LIN {X 101.752,Y 87.486,Z 76.388,A 180.000,B 0.000,C 180.000} C_DIS
LIN {X 101.682,Y 87.454,Z 76.385,A 180.000,B 0.000,C 180.000} C_DIS
LIN {X 101.612,Y 87.423,Z 76.382,A 180.000,B 0.000,C 180.000} C_DIS
LIN {X 101.541,Y 87.395,Z 76.380,A 180.000,B 0.000,C 180.000} C_DIS
LIN {X 101.323,Y 87.307,Z 76.371,A 180.000,B 0.000,C 180.000} C_DIS
LIN {X 101.250,Y 87.278,Z 76.369,A 180.000,B 0.000,C 180.000} C_DIS
LIN {X 101.178,Y 87.250,Z 76.366,A 180.000,B 0.000,C 180.000} C_DIS
LIN {X 101.106,Y 87.223,Z 76.363,A 180.000,B 0.000,C 180.000} C_DIS
LIN {X 101.033,Y 87.198,Z 76.361,A 180.000,B 0.000,C 180.000} C_DIS
LIN {X 100.961,Y 87.173,Z 76.358,A 180.000,B 0.000,C 180.000} C_DIS
LIN {X 100.886,Y 87.148,Z 76.355,A 180.000,B 0.000,C 180.000} C_DIS
LIN {X 100.591,Y 87.048,Z 76.344,A 180.000,B 0.000,C 180.000} C_DIS
LIN {X 100.518,Y 87.024,Z 76.342,A 180.000,B 0.000,C 180.000} C_DIS
LIN {X 100.445,Y 87.002,Z 76.339,A 180.000,B 0.000,C 180.000} C_DIS
LIN {X 100.371,Y 86.981,Z 76.336,A 180.000,B 0.000,C 180.000} C_DIS
LIN {X 100.220,Y 86.940,Z 76.331,A 180.000,B 0.000,C 180.000} C_DIS
LIN {X 100.070,Y 86.898,Z 76.325,A 180.000,B 0.000,C 180.000} C_DIS
LIN {X 99.995,Y 86.878,Z 76.323,A 180.000,B 0.000,C 180.000} C_DIS
LIN {X 99.920,Y 86.860,Z 76.320,A 180.000,B 0.000,C 180.000} C_DIS
LIN {X 99.845,Y 86.843,Z 76.317,A 180.000,B 0.000,C 180.000} C_DIS
LIN {X 99.769,Y 86.827,Z 76.315,A 180.000,B 0.000,C 180.000} C_DIS
LIN {X 99.615,Y 86.794,Z 76.309,A 180.000,B 0.000,C 180.000} C_DIS
LIN {X 99.539,Y 86.777,Z 76.306,A 180.000,B 0.000,C 180.000} C_DIS
LIN {X 99.462,Y 86.760,Z 76.304,A 180.000,B 0.000,C 180.000} C_DIS
LIN {X 99.386,Y 86.745,Z 76.301,A 180.000,B 0.000,C 180.000} C_DIS
LIN {X 99.311,Y 86.729,Z 76.298,A 180.000,B 0.000,C 180.000} C_DIS
LIN {X 99.235,Y 86.716,Z 76.295,A 180.000,B 0.000,C 180.000} C_DIS
LIN {X 99.159,Y 86.703,Z 76.293,A 180.000,B 0.000,C 180.000} C_DIS
LIN {X 99.004,Y 86.679,Z 76.287,A 180.000,B 0.000,C 180.000} C_DIS
LIN {X 98.848,Y 86.654,Z 76.282,A 180.000,B 0.000,C 180.000} C_DIS
LIN {X 98.772,Y 86.643,Z 76.279,A 180.000,B 0.000,C 180.000} C_DIS
LIN {X 98.696,Y 86.633,Z 76.276,A 180.000,B 0.000,C 180.000} C_DIS
LIN {X 98.619,Y 86.625,Z 76.274,A 180.000,B 0.000,C 180.000} C_DIS
LIN {X 98.543,Y 86.617,Z 76.271,A 180.000,B 0.000,C 180.000} C_DIS
LIN {X 98.386,Y 86.602,Z 76.266,A 180.000,B 0.000,C 180.000} C_DIS
LIN {X 98.308,Y 86.594,Z 76.263,A 180.000,B 0.000,C 180.000} C_DIS
LIN {X 98.230,Y 86.586,Z 76.260,A 180.000,B 0.000,C 180.000} C_DIS
LIN {X 98.153,Y 86.580,Z 76.257,A 180.000,B 0.000,C 180.000} C_DIS
LIN {X 98.076,Y 86.574,Z 76.255,A 180.000,B 0.000,C 180.000} C_DIS
LIN {X 97.999,Y 86.569,Z 76.252,A 180.000,B 0.000,C 180.000} C_DIS
LIN {X 97.921,Y 86.565,Z 76.249,A 180.000,B 0.000,C 180.000} C_DIS
LIN {X 97.765,Y 86.558,Z 76.244,A 180.000,B 0.000,C 180.000} C_DIS
LIN {X 97.608,Y 86.551,Z 76.238,A 180.000,B 0.000,C 180.000} C_DIS
LIN {X 97.531,Y 86.548,Z 76.236,A 180.000,B 0.000,C 180.000} C_DIS
LIN {X 97.453,Y 86.547,Z 76.233,A 180.000,B 0.000,C 180.000} C_DIS
LIN {X 97.375,Y 86.548,Z 76.230,A 180.000,B 0.000,C 180.000} C_DIS
LIN {X 97.298,Y 86.549,Z 76.228,A 180.000,B 0.000,C 180.000} C_DIS
LIN {X 97.141,Y 86.551,Z 76.222,A 180.000,B 0.000,C 180.000} C_DIS
LIN {X 97.063,Y 86.552,Z 76.219,A 180.000,B 0.000,C 180.000} C_DIS
LIN {X 96.984,Y 86.553,Z 76.217,A 180.000,B 0.000,C 180.000} C_DIS
LIN {X 96.906,Y 86.556,Z 76.214,A 180.000,B 0.000,C 180.000} C_DIS
LIN {X 96.829,Y 86.559,Z 76.211,A 180.000,B 0.000,C 180.000} C_DIS
LIN {X 96.751,Y 86.563,Z 76.208,A 180.000,B 0.000,C 180.000} C_DIS
LIN {X 96.674,Y 86.568,Z 76.206,A 180.000,B 0.000,C 180.000} C_DIS
LIN {X 96.518,Y 86.579,Z 76.200,A 180.000,B 0.000,C 180.000} C_DIS
LIN {X 96.361,Y 86.590,Z 76.195,A 180.000,B 0.000,C 180.000} C_DIS
LIN {X 96.284,Y 86.595,Z 76.192,A 180.000,B 0.000,C 180.000} C_DIS
LIN {X 96.206,Y 86.603,Z 76.189,A 180.000,B 0.000,C 180.000} C_DIS
LIN {X 96.129,Y 86.613,Z 76.187,A 180.000,B 0.000,C 180.000} C_DIS
LIN {X 95.973,Y 86.632,Z 76.181,A 180.000,B 0.000,C 180.000} C_DIS
LIN {X 95.895,Y 86.642,Z 76.179,A 180.000,B 0.000,C 180.000} C_DIS
LIN {X 95.818,Y 86.652,Z 76.176,A 180.000,B 0.000,C 180.000} C_DIS
LIN {X 95.740,Y 86.662,Z 76.173,A 180.000,B 0.000,C 180.000} C_DIS
LIN {X 95.663,Y 86.674,Z 76.171,A 180.000,B 0.000,C 180.000} C_DIS
LIN {X 95.586,Y 86.687,Z 76.168,A 180.000,B 0.000,C 180.000} C_DIS
LIN {X 95.509,Y 86.701,Z 76.166,A 180.000,B 0.000,C 180.000} C_DIS
LIN {X 95.355,Y 86.729,Z 76.160,A 180.000,B 0.000,C 180.000} C_DIS
LIN {X 95.278,Y 86.743,Z 76.158,A 180.000,B 0.000,C 180.000} C_DIS
LIN {X 95.200,Y 86.757,Z 76.155,A 180.000,B 0.000,C 180.000} C_DIS
LIN {X 95.123,Y 86.771,Z 76.153,A 180.000,B 0.000,C 180.000} C_DIS
LIN {X 94.970,Y 86.803,Z 76.148,A 180.000,B 0.000,C 180.000} C_DIS
LIN {X 94.819,Y 86.839,Z 76.143,A 180.000,B 0.000,C 180.000} C_DIS
LIN {X 94.667,Y 86.876,Z 76.138,A 180.000,B 0.000,C 180.000} C_DIS
LIN {X 94.514,Y 86.914,Z 76.133,A 180.000,B 0.000,C 180.000} C_DIS
LIN {X 94.364,Y 86.957,Z 76.128,A 180.000,B 0.000,C 180.000} C_DIS
LIN {X 94.214,Y 87.002,Z 76.124,A 180.000,B 0.000,C 180.000} C_DIS
LIN {X 94.064,Y 87.048,Z 76.119,A 180.000,B 0.000,C 180.000} C_DIS
LIN {X 93.913,Y 87.094,Z 76.115,A 180.000,B 0.000,C 180.000} C_DIS
LIN {X 93.765,Y 87.143,Z 76.110,A 180.000,B 0.000,C 180.000} C_DIS
LIN {X 93.618,Y 87.197,Z 76.106,A 180.000,B 0.000,C 180.000} C_DIS
LIN {X 93.471,Y 87.251,Z 76.102,A 180.000,B 0.000,C 180.000} C_DIS
LIN {X 93.325,Y 87.305,Z 76.097,A 180.000,B 0.000,C 180.000} C_DIS
LIN {X 93.180,Y 87.366,Z 76.093,A 180.000,B 0.000,C 180.000} C_DIS
LIN {X 93.035,Y 87.429,Z 76.089,A 180.000,B 0.000,C 180.000} C_DIS
LIN {X 92.891,Y 87.491,Z 76.085,A 180.000,B 0.000,C 180.000} C_DIS
LIN {X 92.748,Y 87.555,Z 76.081,A 180.000,B 0.000,C 180.000} C_DIS
LIN {X 92.606,Y 87.622,Z 76.077,A 180.000,B 0.000,C 180.000} C_DIS
LIN {X 92.465,Y 87.692,Z 76.073,A 180.000,B 0.000,C 180.000} C_DIS
LIN {X 92.325,Y 87.763,Z 76.070,A 180.000,B 0.000,C 180.000} C_DIS
LIN {X 92.185,Y 87.834,Z 76.066,A 180.000,B 0.000,C 180.000} C_DIS
LIN {X 92.048,Y 87.911,Z 76.063,A 180.000,B 0.000,C 180.000} C_DIS
LIN {X 91.912,Y 87.989,Z 76.059,A 180.000,B 0.000,C 180.000} C_DIS
LIN {X 91.776,Y 88.068,Z 76.056,A 180.000,B 0.000,C 180.000} C_DIS
LIN {X 91.641,Y 88.148,Z 76.052,A 180.000,B 0.000,C 180.000} C_DIS
LIN {X 91.508,Y 88.232,Z 76.049,A 180.000,B 0.000,C 180.000} C_DIS
LIN {X 91.376,Y 88.318,Z 76.046,A 180.000,B 0.000,C 180.000} C_DIS
LIN {X 91.245,Y 88.404,Z 76.043,A 180.000,B 0.000,C 180.000} C_DIS
LIN {X 91.113,Y 88.491,Z 76.040,A 180.000,B 0.000,C 180.000} C_DIS
LIN {X 90.986,Y 88.583,Z 76.037,A 180.000,B 0.000,C 180.000} C_DIS
LIN {X 90.860,Y 88.677,Z 76.035,A 180.000,B 0.000,C 180.000} C_DIS
LIN {X 90.734,Y 88.770,Z 76.032,A 180.000,B 0.000,C 180.000} C_DIS
LIN {X 90.609,Y 88.866,Z 76.029,A 180.000,B 0.000,C 180.000} C_DIS
LIN {X 90.366,Y 89.066,Z 76.025,A 180.000,B 0.000,C 180.000} C_DIS
LIN {X 90.125,Y 89.268,Z 76.020,A 180.000,B 0.000,C 180.000} C_DIS
LIN {X 89.894,Y 89.482,Z 76.016,A 180.000,B 0.000,C 180.000} C_DIS
LIN {X 89.666,Y 89.700,Z 76.013,A 180.000,B 0.000,C 180.000} C_DIS
LIN {X 89.449,Y 89.927,Z 76.009,A 180.000,B 0.000,C 180.000} C_DIS
LIN {X 89.232,Y 90.156,Z 76.007,A 180.000,B 0.000,C 180.000} C_DIS
LIN {X 89.028,Y 90.395,Z 76.004,A 180.000,B 0.000,C 180.000} C_DIS
LIN {X 88.826,Y 90.638,Z 76.003,A 180.000,B 0.000,C 180.000} C_DIS
LIN {X 88.637,Y 90.889,Z 76.001,A 180.000,B 0.000,C 180.000} C_DIS
LIN {X 88.449,Y 91.142,Z 76.000,A 180.000,B 0.000,C 180.000} C_DIS
LIN {X 88.273,Y 91.403,Z 76.000,A 180.000,B 0.000,C 180.000} C_DIS
LIN {X 88.220,Y 91.484,Z 76.000,A 180.000,B 0.000,C 180.000} C_DIS
; Cutting Move Starts
LIN {X 88.186,Y 91.533,Z 76.000,A 180.000,B 0.000,C 180.000} C_DIS
LIN {X 88.137,Y 91.609,Z 76.000,A 180.000,B 0.000,C 180.000} C_DIS
LIN {X 88.075,Y 91.712,Z 76.000,A 180.000,B 0.000,C 180.000} C_DIS
LIN {X 87.958,Y 91.910,Z 76.000,A 180.000,B 0.000,C 180.000} C_DIS
LIN {X 87.864,Y 92.070,Z 76.000,A 180.000,B 0.000,C 180.000} C_DIS
LIN {X 87.779,Y 92.224,Z 76.000,A 180.000,B 0.000,C 180.000} C_DIS
LIN {X 87.766,Y 92.249,Z 76.000,A 180.000,B 0.000,C 180.000} C_DIS
LIN {X 87.674,Y 92.427,Z 76.000,A 180.000,B 0.000,C 180.000} C_DIS
LIN {X 87.581,Y 92.606,Z 76.000,A 180.000,B 0.000,C 180.000} C_DIS
LIN {X 87.494,Y 92.785,Z 76.000,A 180.000,B 0.000,C 180.000} C_DIS
LIN {X 87.334,Y 93.142,Z 76.000,A 180.000,B 0.000,C 180.000} C_DIS
LIN {X 87.260,Y 93.321,Z 76.000,A 180.000,B 0.000,C 180.000} C_DIS
LIN {X 87.243,Y 93.365,Z 76.000,A 180.000,B 0.000,C 180.000} C_DIS
LIN {X 87.191,Y 93.500,Z 76.000,A 180.000,B 0.000,C 180.000} C_DIS
LIN {X 87.123,Y 93.679,Z 76.000,A 180.000,B 0.000,C 180.000} C_DIS
LIN {X 87.064,Y 93.833,Z 76.000,A 180.000,B 0.000,C 180.000} C_DIS
LIN {X 87.055,Y 93.857,Z 76.000,A 180.000,B 0.000,C 180.000} C_DIS
LIN {X 86.997,Y 94.036,Z 76.000,A 180.000,B 0.000,C 180.000} C_DIS
LIN {X 86.940,Y 94.215,Z 76.000,A 180.000,B 0.000,C 180.000} C_DIS
LIN {X 86.885,Y 94.388,Z 76.000,A 180.000,B 0.000,C 180.000} C_DIS
LIN {X 86.884,Y 94.394,Z 76.000,A 180.000,B 0.000,C 180.000} C_DIS
LIN {X 86.836,Y 94.573,Z 76.000,A 180.000,B 0.000,C 180.000} C_DIS
LIN {X 86.790,Y 94.751,Z 76.000,A 180.000,B 0.000,C 180.000} C_DIS
LIN {X 86.744,Y 94.930,Z 76.000,A 180.000,B 0.000,C 180.000} C_DIS
LIN {X 86.707,Y 95.079,Z 76.000,A 180.000,B 0.000,C 180.000} C_DIS
LIN {X 86.700,Y 95.109,Z 76.000,A 180.000,B 0.000,C 180.000} C_DIS
LIN {X 86.664,Y 95.288,Z 76.000,A 180.000,B 0.000,C 180.000} C_DIS
LIN {X 86.629,Y 95.466,Z 76.000,A 180.000,B 0.000,C 180.000} C_DIS
LIN {X 86.595,Y 95.645,Z 76.000,A 180.000,B 0.000,C 180.000} C_DIS
LIN {X 86.569,Y 95.824,Z 76.000,A 180.000,B 0.000,C 180.000} C_DIS
LIN {X 86.528,Y 96.116,Z 76.000,A 180.000,B 0.000,C 180.000} C_DIS
LIN {X 86.519,Y 96.181,Z 76.000,A 180.000,B 0.000,C 180.000} C_DIS
LIN {X 86.498,Y 96.360,Z 76.000,A 180.000,B 0.000,C 180.000} C_DIS
LIN {X 86.483,Y 96.539,Z 76.000,A 180.000,B 0.000,C 180.000} C_DIS
LIN {X 86.468,Y 96.718,Z 76.000,A 180.000,B 0.000,C 180.000} C_DIS
LIN {X 86.455,Y 96.897,Z 76.000,A 180.000,B 0.000,C 180.000} C_DIS
LIN {X 86.449,Y 97.075,Z 76.000,A 180.000,B 0.000,C 180.000} C_DIS
LIN {X 86.444,Y 97.254,Z 76.000,A 180.000,B 0.000,C 180.000} C_DIS
LIN {X 86.440,Y 97.433,Z 76.000,A 180.000,B 0.000,C 180.000} C_DIS
LIN {X 86.440,Y 97.612,Z 76.000,A 180.000,B 0.000,C 180.000} C_DIS
LIN {X 86.445,Y 97.790,Z 76.000,A 180.000,B 0.000,C 180.000} C_DIS
LIN {X 86.450,Y 97.969,Z 76.000,A 180.000,B 0.000,C 180.000} C_DIS
LIN {X 86.457,Y 98.148,Z 76.000,A 180.000,B 0.000,C 180.000} C_DIS
LIN {X 86.472,Y 98.327,Z 76.000,A 180.000,B 0.000,C 180.000} C_DIS
LIN {X 86.487,Y 98.505,Z 76.000,A 180.000,B 0.000,C 180.000} C_DIS
LIN {X 86.503,Y 98.684,Z 76.000,A 180.000,B 0.000,C 180.000} C_DIS
LIN {X 86.525,Y 98.863,Z 76.000,A 180.000,B 0.000,C 180.000} C_DIS
LIN {X 86.528,Y 98.884,Z 76.000,A 180.000,B 0.000,C 180.000} C_DIS
LIN {X 86.575,Y 99.221,Z 76.000,A 180.000,B 0.000,C 180.000} C_DIS
LIN {X 86.603,Y 99.399,Z 76.000,A 180.000,B 0.000,C 180.000} C_DIS
LIN {X 86.638,Y 99.578,Z 76.000,A 180.000,B 0.000,C 180.000} C_DIS
LIN {X 86.673,Y 99.757,Z 76.000,A 180.000,B 0.000,C 180.000} C_DIS
LIN {X 86.707,Y 99.921,Z 76.000,A 180.000,B 0.000,C 180.000} C_DIS
LIN {X 86.710,Y 99.936,Z 76.000,A 180.000,B 0.000,C 180.000} C_DIS
LIN {X 86.755,Y 100.114,Z 76.000,A 180.000,B 0.000,C 180.000} C_DIS
LIN {X 86.848,Y 100.472,Z 76.000,A 180.000,B 0.000,C 180.000} C_DIS
LIN {X 86.885,Y 100.612,Z 76.000,A 180.000,B 0.000,C 180.000} C_DIS
LIN {X 86.897,Y 100.651,Z 76.000,A 180.000,B 0.000,C 180.000} C_DIS
LIN {X 86.954,Y 100.829,Z 76.000,A 180.000,B 0.000,C 180.000} C_DIS
LIN {X 87.011,Y 101.008,Z 76.000,A 180.000,B 0.000,C 180.000} C_DIS
LIN {X 87.064,Y 101.167,Z 76.000,A 180.000,B 0.000,C 180.000} C_DIS
LIN {X 87.071,Y 101.187,Z 76.000,A 180.000,B 0.000,C 180.000} C_DIS
LIN {X 87.140,Y 101.366,Z 76.000,A 180.000,B 0.000,C 180.000} C_DIS
LIN {X 87.208,Y 101.545,Z 76.000,A 180.000,B 0.000,C 180.000} C_DIS
LIN {X 87.243,Y 101.635,Z 76.000,A 180.000,B 0.000,C 180.000} C_DIS
LIN {X 87.278,Y 101.723,Z 76.000,A 180.000,B 0.000,C 180.000} C_DIS
LIN {X 87.354,Y 101.902,Z 76.000,A 180.000,B 0.000,C 180.000} C_DIS
LIN {X 87.434,Y 102.081,Z 76.000,A 180.000,B 0.000,C 180.000} C_DIS
LIN {X 87.515,Y 102.260,Z 76.000,A 180.000,B 0.000,C 180.000} C_DIS
LIN {X 87.601,Y 102.431,Z 76.000,A 180.000,B 0.000,C 180.000} C_DIS
LIN {X 87.697,Y 102.617,Z 76.000,A 180.000,B 0.000,C 180.000} C_DIS
LIN {X 87.779,Y 102.776,Z 76.000,A 180.000,B 0.000,C 180.000} C_DIS
LIN {X 87.790,Y 102.796,Z 76.000,A 180.000,B 0.000,C 180.000} C_DIS
LIN {X 87.890,Y 102.975,Z 76.000,A 180.000,B 0.000,C 180.000} C_DIS
LIN {X 88.101,Y 103.332,Z 76.000,A 180.000,B 0.000,C 180.000} C_DIS
LIN {X 88.137,Y 103.391,Z 76.000,A 180.000,B 0.000,C 180.000} C_DIS
LIN {X 88.216,Y 103.511,Z 76.000,A 180.000,B 0.000,C 180.000} C_DIS
LIN {X 88.336,Y 103.690,Z 76.000,A 180.000,B 0.000,C 180.000} C_DIS
LIN {X 88.457,Y 103.869,Z 76.000,A 180.000,B 0.000,C 180.000} C_DIS
LIN {X 88.494,Y 103.920,Z 76.000,A 180.000,B 0.000,C 180.000} C_DIS
LIN {X 88.588,Y 104.047,Z 76.000,A 180.000,B 0.000,C 180.000} C_DIS
LIN {X 88.722,Y 104.226,Z 76.000,A 180.000,B 0.000,C 180.000} C_DIS
LIN {X 88.852,Y 104.397,Z 76.000,A 180.000,B 0.000,C 180.000} C_DIS
LIN {X 88.858,Y 104.405,Z 76.000,A 180.000,B 0.000,C 180.000} C_DIS
LIN {X 89.007,Y 104.584,Z 76.000,A 180.000,B 0.000,C 180.000} C_DIS
LIN {X 89.158,Y 104.762,Z 76.000,A 180.000,B 0.000,C 180.000} C_DIS
LIN {X 89.209,Y 104.823,Z 76.000,A 180.000,B 0.000,C 180.000} C_DIS
LIN {X 89.319,Y 104.941,Z 76.000,A 180.000,B 0.000,C 180.000} C_DIS
LIN {X 89.388,Y 105.015,Z 76.000,A 180.000,B 0.000,C 180.000} C_DIS
LIN {X 89.567,Y 105.204,Z 76.000,A 180.000,B 0.000,C 180.000} C_DIS
LIN {X 89.656,Y 105.299,Z 76.000,A 180.000,B 0.000,C 180.000} C_DIS
LIN {X 89.746,Y 105.388,Z 76.000,A 180.000,B 0.000,C 180.000} C_DIS
LIN {X 89.925,Y 105.557,Z 76.000,A 180.000,B 0.000,C 180.000} C_DIS
LIN {X 90.030,Y 105.656,Z 76.000,A 180.000,B 0.000,C 180.000} C_DIS
LIN {X 90.103,Y 105.725,Z 76.000,A 180.000,B 0.000,C 180.000} C_DIS
LIN {X 90.232,Y 105.835,Z 76.000,A 180.000,B 0.000,C 180.000} C_DIS
LIN {X 90.461,Y 106.029,Z 76.000,A 180.000,B 0.000,C 180.000} C_DIS
LIN {X 90.640,Y 106.177,Z 76.000,A 180.000,B 0.000,C 180.000} C_DIS
LIN {X 90.660,Y 106.193,Z 76.000,A 180.000,B 0.000,C 180.000} C_DIS
LIN {X 90.818,Y 106.312,Z 76.000,A 180.000,B 0.000,C 180.000} C_DIS
LIN {X 90.997,Y 106.447,Z 76.000,A 180.000,B 0.000,C 180.000} C_DIS
LIN {X 91.140,Y 106.550,Z 76.000,A 180.000,B 0.000,C 180.000} C_DIS
LIN {X 91.176,Y 106.574,Z 76.000,A 180.000,B 0.000,C 180.000} C_DIS
LIN {X 91.408,Y 106.729,Z 76.000,A 180.000,B 0.000,C 180.000} C_DIS
LIN {X 91.533,Y 106.813,Z 76.000,A 180.000,B 0.000,C 180.000} C_DIS
LIN {X 91.684,Y 106.908,Z 76.000,A 180.000,B 0.000,C 180.000} C_DIS
LIN {X 91.712,Y 106.925,Z 76.000,A 180.000,B 0.000,C 180.000} C_DIS
LIN {X 91.891,Y 107.031,Z 76.000,A 180.000,B 0.000,C 180.000} C_DIS
LIN {X 92.070,Y 107.136,Z 76.000,A 180.000,B 0.000,C 180.000} C_DIS
LIN {X 92.249,Y 107.234,Z 76.000,A 180.000,B 0.000,C 180.000} C_DIS
LIN {X 92.427,Y 107.327,Z 76.000,A 180.000,B 0.000,C 180.000} C_DIS
LIN {X 92.606,Y 107.419,Z 76.000,A 180.000,B 0.000,C 180.000} C_DIS
LIN {X 92.657,Y 107.444,Z 76.000,A 180.000,B 0.000,C 180.000} C_DIS
LIN {X 92.785,Y 107.504,Z 76.000,A 180.000,B 0.000,C 180.000} C_DIS
LIN {X 92.964,Y 107.585,Z 76.000,A 180.000,B 0.000,C 180.000} C_DIS
LIN {X 93.142,Y 107.665,Z 76.000,A 180.000,B 0.000,C 180.000} C_DIS
LIN {X 93.321,Y 107.742,Z 76.000,A 180.000,B 0.000,C 180.000} C_DIS
LIN {X 93.477,Y 107.802,Z 76.000,A 180.000,B 0.000,C 180.000} C_DIS
LIN {X 93.679,Y 107.879,Z 76.000,A 180.000,B 0.000,C 180.000} C_DIS
LIN {X 93.857,Y 107.944,Z 76.000,A 180.000,B 0.000,C 180.000} C_DIS
LIN {X 93.970,Y 107.980,Z 76.000,A 180.000,B 0.000,C 180.000} C_DIS
LIN {X 94.036,Y 108.001,Z 76.000,A 180.000,B 0.000,C 180.000} C_DIS
LIN {X 94.394,Y 108.115,Z 76.000,A 180.000,B 0.000,C 180.000} C_DIS
LIN {X 94.546,Y 108.159,Z 76.000,A 180.000,B 0.000,C 180.000} C_DIS
LIN {X 94.930,Y 108.258,Z 76.000,A 180.000,B 0.000,C 180.000} C_DIS
LIN {X 95.109,Y 108.299,Z 76.000,A 180.000,B 0.000,C 180.000} C_DIS
LIN {X 95.466,Y 108.370,Z 76.000,A 180.000,B 0.000,C 180.000} C_DIS
LIN {X 95.645,Y 108.404,Z 76.000,A 180.000,B 0.000,C 180.000} C_DIS
LIN {X 95.824,Y 108.432,Z 76.000,A 180.000,B 0.000,C 180.000} C_DIS
LIN {X 96.181,Y 108.482,Z 76.000,A 180.000,B 0.000,C 180.000} C_DIS
LIN {X 96.360,Y 108.501,Z 76.000,A 180.000,B 0.000,C 180.000} C_DIS
LIN {X 96.718,Y 108.531,Z 76.000,A 180.000,B 0.000,C 180.000} C_DIS
LIN {X 96.897,Y 108.544,Z 76.000,A 180.000,B 0.000,C 180.000} C_DIS
LIN {X 97.075,Y 108.551,Z 76.000,A 180.000,B 0.000,C 180.000} C_DIS
LIN {X 97.433,Y 108.561,Z 76.000,A 180.000,B 0.000,C 180.000} C_DIS
LIN {X 97.612,Y 108.560,Z 76.000,A 180.000,B 0.000,C 180.000} C_DIS
LIN {X 97.969,Y 108.550,Z 76.000,A 180.000,B 0.000,C 180.000} C_DIS
LIN {X 98.148,Y 108.541,Z 76.000,A 180.000,B 0.000,C 180.000} C_DIS
LIN {X 98.327,Y 108.528,Z 76.000,A 180.000,B 0.000,C 180.000} C_DIS
LIN {X 98.684,Y 108.498,Z 76.000,A 180.000,B 0.000,C 180.000} C_DIS
LIN {X 98.863,Y 108.476,Z 76.000,A 180.000,B 0.000,C 180.000} C_DIS
LIN {X 99.221,Y 108.426,Z 76.000,A 180.000,B 0.000,C 180.000} C_DIS
LIN {X 99.399,Y 108.396,Z 76.000,A 180.000,B 0.000,C 180.000} C_DIS
LIN {X 99.578,Y 108.361,Z 76.000,A 180.000,B 0.000,C 180.000} C_DIS
LIN {X 99.757,Y 108.325,Z 76.000,A 180.000,B 0.000,C 180.000} C_DIS
LIN {X 99.936,Y 108.290,Z 76.000,A 180.000,B 0.000,C 180.000} C_DIS
LIN {X 100.114,Y 108.247,Z 76.000,A 180.000,B 0.000,C 180.000} C_DIS
LIN {X 100.472,Y 108.154,Z 76.000,A 180.000,B 0.000,C 180.000} C_DIS
LIN {X 100.651,Y 108.101,Z 76.000,A 180.000,B 0.000,C 180.000} C_DIS
LIN {X 101.008,Y 107.987,Z 76.000,A 180.000,B 0.000,C 180.000} C_DIS
LIN {X 101.030,Y 107.980,Z 76.000,A 180.000,B 0.000,C 180.000} C_DIS
LIN {X 101.187,Y 107.929,Z 76.000,A 180.000,B 0.000,C 180.000} C_DIS
LIN {X 101.366,Y 107.862,Z 76.000,A 180.000,B 0.000,C 180.000} C_DIS
LIN {X 101.545,Y 107.793,Z 76.000,A 180.000,B 0.000,C 180.000} C_DIS
LIN {X 101.723,Y 107.724,Z 76.000,A 180.000,B 0.000,C 180.000} C_DIS
LIN {X 101.902,Y 107.645,Z 76.000,A 180.000,B 0.000,C 180.000} C_DIS
LIN {X 102.081,Y 107.565,Z 76.000,A 180.000,B 0.000,C 180.000} C_DIS
LIN {X 102.260,Y 107.483,Z 76.000,A 180.000,B 0.000,C 180.000} C_DIS
LIN {X 102.343,Y 107.444,Z 76.000,A 180.000,B 0.000,C 180.000} C_DIS
LIN {X 102.438,Y 107.396,Z 76.000,A 180.000,B 0.000,C 180.000} C_DIS
LIN {X 102.692,Y 107.265,Z 76.000,A 180.000,B 0.000,C 180.000} C_DIS
LIN {X 102.796,Y 107.211,Z 76.000,A 180.000,B 0.000,C 180.000} C_DIS
LIN {X 102.975,Y 107.110,Z 76.000,A 180.000,B 0.000,C 180.000} C_DIS
LIN {X 103.153,Y 107.004,Z 76.000,A 180.000,B 0.000,C 180.000} C_DIS
LIN {X 103.316,Y 106.908,Z 76.000,A 180.000,B 0.000,C 180.000} C_DIS
LIN {X 103.332,Y 106.898,Z 76.000,A 180.000,B 0.000,C 180.000} C_DIS
LIN {X 103.511,Y 106.783,Z 76.000,A 180.000,B 0.000,C 180.000} C_DIS
LIN {X 103.690,Y 106.664,Z 76.000,A 180.000,B 0.000,C 180.000} C_DIS
LIN {X 103.860,Y 106.550,Z 76.000,A 180.000,B 0.000,C 180.000} C_DIS
LIN {X 103.869,Y 106.544,Z 76.000,A 180.000,B 0.000,C 180.000} C_DIS
LIN {X 104.047,Y 106.413,Z 76.000,A 180.000,B 0.000,C 180.000} C_DIS
LIN {X 104.226,Y 106.279,Z 76.000,A 180.000,B 0.000,C 180.000} C_DIS
LIN {X 104.340,Y 106.193,Z 76.000,A 180.000,B 0.000,C 180.000} C_DIS
LIN {X 104.405,Y 106.140,Z 76.000,A 180.000,B 0.000,C 180.000} C_DIS
LIN {X 104.557,Y 106.014,Z 76.000,A 180.000,B 0.000,C 180.000} C_DIS
LIN {X 104.715,Y 105.880,Z 76.000,A 180.000,B 0.000,C 180.000} C_DIS
LIN {X 104.768,Y 105.835,Z 76.000,A 180.000,B 0.000,C 180.000} C_DIS
LIN {X 104.941,Y 105.684,Z 76.000,A 180.000,B 0.000,C 180.000} C_DIS
LIN {X 105.160,Y 105.477,Z 76.000,A 180.000,B 0.000,C 180.000} C_DIS
LIN {X 105.299,Y 105.345,Z 76.000,A 180.000,B 0.000,C 180.000} C_DIS
LIN {X 105.344,Y 105.299,Z 76.000,A 180.000,B 0.000,C 180.000} C_DIS
LIN {X 105.513,Y 105.120,Z 76.000,A 180.000,B 0.000,C 180.000} C_DIS
LIN {X 105.656,Y 104.968,Z 76.000,A 180.000,B 0.000,C 180.000} C_DIS
LIN {X 105.681,Y 104.941,Z 76.000,A 180.000,B 0.000,C 180.000} C_DIS
LIN {X 105.835,Y 104.770,Z 76.000,A 180.000,B 0.000,C 180.000} C_DIS
LIN {X 106.014,Y 104.559,Z 76.000,A 180.000,B 0.000,C 180.000} C_DIS
LIN {X 106.142,Y 104.405,Z 76.000,A 180.000,B 0.000,C 180.000} C_DIS
LIN {X 106.193,Y 104.339,Z 76.000,A 180.000,B 0.000,C 180.000} C_DIS
LIN {X 106.412,Y 104.047,Z 76.000,A 180.000,B 0.000,C 180.000} C_DIS
LIN {X 106.543,Y 103.869,Z 76.000,A 180.000,B 0.000,C 180.000} C_DIS
LIN {X 106.550,Y 103.859,Z 76.000,A 180.000,B 0.000,C 180.000} C_DIS
LIN {X 106.664,Y 103.690,Z 76.000,A 180.000,B 0.000,C 180.000} C_DIS
LIN {X 106.784,Y 103.511,Z 76.000,A 180.000,B 0.000,C 180.000} C_DIS
LIN {X 106.899,Y 103.332,Z 76.000,A 180.000,B 0.000,C 180.000} C_DIS
LIN {X 107.110,Y 102.975,Z 76.000,A 180.000,B 0.000,C 180.000} C_DIS
LIN {X 107.210,Y 102.796,Z 76.000,A 180.000,B 0.000,C 180.000} C_DIS
LIN {X 107.265,Y 102.691,Z 76.000,A 180.000,B 0.000,C 180.000} C_DIS
LIN {X 107.396,Y 102.438,Z 76.000,A 180.000,B 0.000,C 180.000} C_DIS
LIN {X 107.444,Y 102.345,Z 76.000,A 180.000,B 0.000,C 180.000} C_DIS
LIN {X 107.485,Y 102.260,Z 76.000,A 180.000,B 0.000,C 180.000} C_DIS
LIN {X 107.566,Y 102.081,Z 76.000,A 180.000,B 0.000,C 180.000} C_DIS
LIN {X 107.646,Y 101.902,Z 76.000,A 180.000,B 0.000,C 180.000} C_DIS
LIN {X 107.722,Y 101.723,Z 76.000,A 180.000,B 0.000,C 180.000} C_DIS
LIN {X 107.792,Y 101.545,Z 76.000,A 180.000,B 0.000,C 180.000} C_DIS
LIN {X 107.860,Y 101.366,Z 76.000,A 180.000,B 0.000,C 180.000} C_DIS
LIN {X 107.929,Y 101.187,Z 76.000,A 180.000,B 0.000,C 180.000} C_DIS
LIN {X 107.980,Y 101.036,Z 76.000,A 180.000,B 0.000,C 180.000} C_DIS
LIN {X 108.046,Y 100.829,Z 76.000,A 180.000,B 0.000,C 180.000} C_DIS
LIN {X 108.103,Y 100.651,Z 76.000,A 180.000,B 0.000,C 180.000} C_DIS
LIN {X 108.152,Y 100.472,Z 76.000,A 180.000,B 0.000,C 180.000} C_DIS
LIN {X 108.245,Y 100.114,Z 76.000,A 180.000,B 0.000,C 180.000} C_DIS
LIN {X 108.290,Y 99.936,Z 76.000,A 180.000,B 0.000,C 180.000} C_DIS
LIN {X 108.327,Y 99.757,Z 76.000,A 180.000,B 0.000,C 180.000} C_DIS
LIN {X 108.362,Y 99.578,Z 76.000,A 180.000,B 0.000,C 180.000} C_DIS
LIN {X 108.397,Y 99.399,Z 76.000,A 180.000,B 0.000,C 180.000} C_DIS
LIN {X 108.425,Y 99.221,Z 76.000,A 180.000,B 0.000,C 180.000} C_DIS
LIN {X 108.450,Y 99.042,Z 76.000,A 180.000,B 0.000,C 180.000} C_DIS
LIN {X 108.475,Y 98.863,Z 76.000,A 180.000,B 0.000,C 180.000} C_DIS
LIN {X 108.497,Y 98.684,Z 76.000,A 180.000,B 0.000,C 180.000} C_DIS
LIN {X 108.513,Y 98.505,Z 76.000,A 180.000,B 0.000,C 180.000} C_DIS
LIN {X 108.528,Y 98.327,Z 76.000,A 180.000,B 0.000,C 180.000} C_DIS
LIN {X 108.543,Y 98.148,Z 76.000,A 180.000,B 0.000,C 180.000} C_DIS
LIN {X 108.550,Y 97.969,Z 76.000,A 180.000,B 0.000,C 180.000} C_DIS
LIN {X 108.555,Y 97.790,Z 76.000,A 180.000,B 0.000,C 180.000} C_DIS
LIN {X 108.560,Y 97.612,Z 76.000,A 180.000,B 0.000,C 180.000} C_DIS
LIN {X 108.560,Y 97.433,Z 76.000,A 180.000,B 0.000,C 180.000} C_DIS
LIN {X 108.556,Y 97.254,Z 76.000,A 180.000,B 0.000,C 180.000} C_DIS
LIN {X 108.551,Y 97.075,Z 76.000,A 180.000,B 0.000,C 180.000} C_DIS
LIN {X 108.545,Y 96.897,Z 76.000,A 180.000,B 0.000,C 180.000} C_DIS
LIN {X 108.532,Y 96.718,Z 76.000,A 180.000,B 0.000,C 180.000} C_DIS
LIN {X 108.517,Y 96.534,Z 76.000,A 180.000,B 0.000,C 180.000} C_DIS
LIN {X 108.502,Y 96.360,Z 76.000,A 180.000,B 0.000,C 180.000} C_DIS
LIN {X 108.481,Y 96.181,Z 76.000,A 180.000,B 0.000,C 180.000} C_DIS
LIN {X 108.456,Y 96.003,Z 76.000,A 180.000,B 0.000,C 180.000} C_DIS
LIN {X 108.431,Y 95.824,Z 76.000,A 180.000,B 0.000,C 180.000} C_DIS
LIN {X 108.405,Y 95.645,Z 76.000,A 180.000,B 0.000,C 180.000} C_DIS
LIN {X 108.371,Y 95.466,Z 76.000,A 180.000,B 0.000,C 180.000} C_DIS
LIN {X 108.336,Y 95.288,Z 76.000,A 180.000,B 0.000,C 180.000} C_DIS
LIN {X 108.300,Y 95.109,Z 76.000,A 180.000,B 0.000,C 180.000} C_DIS
LIN {X 108.256,Y 94.930,Z 76.000,A 180.000,B 0.000,C 180.000} C_DIS
LIN {X 108.210,Y 94.751,Z 76.000,A 180.000,B 0.000,C 180.000} C_DIS
LIN {X 108.159,Y 94.554,Z 76.000,A 180.000,B 0.000,C 180.000} C_DIS
LIN {X 108.116,Y 94.394,Z 76.000,A 180.000,B 0.000,C 180.000} C_DIS
LIN {X 108.060,Y 94.215,Z 76.000,A 180.000,B 0.000,C 180.000} C_DIS
LIN {X 107.980,Y 93.964,Z 76.000,A 180.000,B 0.000,C 180.000} C_DIS
LIN {X 107.945,Y 93.857,Z 76.000,A 180.000,B 0.000,C 180.000} C_DIS
LIN {X 107.877,Y 93.679,Z 76.000,A 180.000,B 0.000,C 180.000} C_DIS
LIN {X 107.802,Y 93.480,Z 76.000,A 180.000,B 0.000,C 180.000} C_DIS
LIN {X 107.740,Y 93.321,Z 76.000,A 180.000,B 0.000,C 180.000} C_DIS
LIN {X 107.666,Y 93.142,Z 76.000,A 180.000,B 0.000,C 180.000} C_DIS
LIN {X 107.506,Y 92.785,Z 76.000,A 180.000,B 0.000,C 180.000} C_DIS
LIN {X 107.444,Y 92.655,Z 76.000,A 180.000,B 0.000,C 180.000} C_DIS
LIN {X 107.419,Y 92.606,Z 76.000,A 180.000,B 0.000,C 180.000} C_DIS
LIN {X 107.265,Y 92.309,Z 76.000,A 180.000,B 0.000,C 180.000} C_DIS
LIN {X 107.234,Y 92.249,Z 76.000,A 180.000,B 0.000,C 180.000} C_DIS
LIN {X 107.136,Y 92.070,Z 76.000,A 180.000,B 0.000,C 180.000} C_DIS
LIN {X 107.086,Y 91.986,Z 76.000,A 180.000,B 0.000,C 180.000} C_DIS
LIN {X 106.908,Y 91.683,Z 76.000,A 180.000,B 0.000,C 180.000} C_DIS
LIN {X 106.814,Y 91.533,Z 76.000,A 180.000,B 0.000,C 180.000} C_DIS
LIN {X 106.694,Y 91.355,Z 76.000,A 180.000,B 0.000,C 180.000} C_DIS
LIN {X 106.574,Y 91.176,Z 76.000,A 180.000,B 0.000,C 180.000} C_DIS
LIN {X 106.550,Y 91.141,Z 76.000,A 180.000,B 0.000,C 180.000} C_DIS
LIN {X 106.446,Y 90.997,Z 76.000,A 180.000,B 0.000,C 180.000} C_DIS
LIN {X 106.371,Y 90.898,Z 76.000,A 180.000,B 0.000,C 180.000} C_DIS
LIN {X 106.193,Y 90.661,Z 76.000,A 180.000,B 0.000,C 180.000} C_DIS
LIN {X 106.177,Y 90.640,Z 76.000,A 180.000,B 0.000,C 180.000} C_DIS
LIN {X 106.030,Y 90.461,Z 76.000,A 180.000,B 0.000,C 180.000} C_DIS
LIN {X 105.835,Y 90.230,Z 76.000,A 180.000,B 0.000,C 180.000} C_DIS
LIN {X 105.723,Y 90.103,Z 76.000,A 180.000,B 0.000,C 180.000} C_DIS
LIN {X 105.656,Y 90.032,Z 76.000,A 180.000,B 0.000,C 180.000} C_DIS
LIN {X 105.555,Y 89.925,Z 76.000,A 180.000,B 0.000,C 180.000} C_DIS
LIN {X 105.386,Y 89.746,Z 76.000,A 180.000,B 0.000,C 180.000} C_DIS
LIN {X 105.299,Y 89.655,Z 76.000,A 180.000,B 0.000,C 180.000} C_DIS
LIN {X 105.207,Y 89.567,Z 76.000,A 180.000,B 0.000,C 180.000} C_DIS
LIN {X 104.941,Y 89.316,Z 76.000,A 180.000,B 0.000,C 180.000} C_DIS
LIN {X 104.821,Y 89.209,Z 76.000,A 180.000,B 0.000,C 180.000} C_DIS
LIN {X 104.584,Y 89.009,Z 76.000,A 180.000,B 0.000,C 180.000} C_DIS
LIN {X 104.405,Y 88.860,Z 76.000,A 180.000,B 0.000,C 180.000} C_DIS
LIN {X 104.396,Y 88.852,Z 76.000,A 180.000,B 0.000,C 180.000} C_DIS
LIN {X 104.226,Y 88.721,Z 76.000,A 180.000,B 0.000,C 180.000} C_DIS
LIN {X 104.047,Y 88.587,Z 76.000,A 180.000,B 0.000,C 180.000} C_DIS
LIN {X 103.924,Y 88.494,Z 76.000,A 180.000,B 0.000,C 180.000} C_DIS
LIN {X 103.869,Y 88.456,Z 76.000,A 180.000,B 0.000,C 180.000} C_DIS
LIN {X 103.690,Y 88.336,Z 76.000,A 180.000,B 0.000,C 180.000} C_DIS
LIN {X 103.511,Y 88.217,Z 76.000,A 180.000,B 0.000,C 180.000} C_DIS
LIN {X 103.387,Y 88.137,Z 76.000,A 180.000,B 0.000,C 180.000} C_DIS
LIN {X 103.332,Y 88.102,Z 76.000,A 180.000,B 0.000,C 180.000} C_DIS
LIN {X 103.153,Y 87.996,Z 76.000,A 180.000,B 0.000,C 180.000} C_DIS
LIN {X 102.975,Y 87.890,Z 76.000,A 180.000,B 0.000,C 180.000} C_DIS
LIN {X 102.796,Y 87.789,Z 76.000,A 180.000,B 0.000,C 180.000} C_DIS
LIN {X 102.778,Y 87.779,Z 76.000,A 180.000,B 0.000,C 180.000} C_DIS
LIN {X 102.432,Y 87.601,Z 76.000,A 180.000,B 0.000,C 180.000} C_DIS
LIN {X 102.260,Y 87.517,Z 76.000,A 180.000,B 0.000,C 180.000} C_DIS
LIN {X 102.081,Y 87.435,Z 76.000,A 180.000,B 0.000,C 180.000} C_DIS
LIN {X 101.902,Y 87.355,Z 76.000,A 180.000,B 0.000,C 180.000} C_DIS
LIN {X 101.723,Y 87.276,Z 76.000,A 180.000,B 0.000,C 180.000} C_DIS
LIN {X 101.640,Y 87.243,Z 76.000,A 180.000,B 0.000,C 180.000} C_DIS
LIN {X 101.366,Y 87.138,Z 76.000,A 180.000,B 0.000,C 180.000} C_DIS
LIN {X 101.187,Y 87.071,Z 76.000,A 180.000,B 0.000,C 180.000} C_DIS
LIN {X 101.166,Y 87.064,Z 76.000,A 180.000,B 0.000,C 180.000} C_DIS
LIN {X 101.008,Y 87.013,Z 76.000,A 180.000,B 0.000,C 180.000} C_DIS
LIN {X 100.609,Y 86.885,Z 76.000,A 180.000,B 0.000,C 180.000} C_DIS
LIN {X 100.472,Y 86.846,Z 76.000,A 180.000,B 0.000,C 180.000} C_DIS
LIN {X 100.114,Y 86.753,Z 76.000,A 180.000,B 0.000,C 180.000} C_DIS
LIN {X 99.936,Y 86.710,Z 76.000,A 180.000,B 0.000,C 180.000} C_DIS
LIN {X 99.917,Y 86.707,Z 76.000,A 180.000,B 0.000,C 180.000} C_DIS
LIN {X 99.578,Y 86.639,Z 76.000,A 180.000,B 0.000,C 180.000} C_DIS
LIN {X 99.399,Y 86.604,Z 76.000,A 180.000,B 0.000,C 180.000} C_DIS
LIN {X 99.221,Y 86.574,Z 76.000,A 180.000,B 0.000,C 180.000} C_DIS
LIN {X 98.863,Y 86.524,Z 76.000,A 180.000,B 0.000,C 180.000} C_DIS
LIN {X 98.684,Y 86.502,Z 76.000,A 180.000,B 0.000,C 180.000} C_DIS
LIN {X 98.327,Y 86.472,Z 76.000,A 180.000,B 0.000,C 180.000} C_DIS
LIN {X 98.148,Y 86.459,Z 76.000,A 180.000,B 0.000,C 180.000} C_DIS
LIN {X 97.969,Y 86.450,Z 76.000,A 180.000,B 0.000,C 180.000} C_DIS
LIN {X 97.612,Y 86.440,Z 76.000,A 180.000,B 0.000,C 180.000} C_DIS
LIN {X 97.433,Y 86.439,Z 76.000,A 180.000,B 0.000,C 180.000} C_DIS
LIN {X 97.075,Y 86.449,Z 76.000,A 180.000,B 0.000,C 180.000} C_DIS
LIN {X 96.897,Y 86.456,Z 76.000,A 180.000,B 0.000,C 180.000} C_DIS
LIN {X 96.718,Y 86.469,Z 76.000,A 180.000,B 0.000,C 180.000} C_DIS
LIN {X 96.360,Y 86.499,Z 76.000,A 180.000,B 0.000,C 180.000} C_DIS
LIN {X 96.181,Y 86.518,Z 76.000,A 180.000,B 0.000,C 180.000} C_DIS
LIN {X 95.824,Y 86.568,Z 76.000,A 180.000,B 0.000,C 180.000} C_DIS
LIN {X 95.645,Y 86.596,Z 76.000,A 180.000,B 0.000,C 180.000} C_DIS
LIN {X 95.466,Y 86.630,Z 76.000,A 180.000,B 0.000,C 180.000} C_DIS
LIN {X 95.083,Y 86.707,Z 76.000,A 180.000,B 0.000,C 180.000} C_DIS
LIN {X 94.930,Y 86.742,Z 76.000,A 180.000,B 0.000,C 180.000} C_DIS
LIN {X 94.573,Y 86.834,Z 76.000,A 180.000,B 0.000,C 180.000} C_DIS
LIN {X 94.394,Y 86.885,Z 76.000,A 180.000,B 0.000,C 180.000} C_DIS
LIN {X 94.036,Y 86.999,Z 76.000,A 180.000,B 0.000,C 180.000} C_DIS
LIN {X 93.857,Y 87.056,Z 76.000,A 180.000,B 0.000,C 180.000} C_DIS
LIN {X 93.834,Y 87.064,Z 76.000,A 180.000,B 0.000,C 180.000} C_DIS
LIN {X 93.679,Y 87.121,Z 76.000,A 180.000,B 0.000,C 180.000} C_DIS
LIN {X 93.360,Y 87.243,Z 76.000,A 180.000,B 0.000,C 180.000} C_DIS
LIN {X 93.321,Y 87.258,Z 76.000,A 180.000,B 0.000,C 180.000} C_DIS
LIN {X 93.142,Y 87.335,Z 76.000,A 180.000,B 0.000,C 180.000} C_DIS
LIN {X 92.949,Y 87.422,Z 76.000,A 180.000,B 0.000,C 180.000} C_DIS
LIN {X 92.785,Y 87.496,Z 76.000,A 180.000,B 0.000,C 180.000} C_DIS
LIN {X 92.606,Y 87.581,Z 76.000,A 180.000,B 0.000,C 180.000} C_DIS
LIN {X 92.568,Y 87.601,Z 76.000,A 180.000,B 0.000,C 180.000} C_DIS
LIN {X 92.222,Y 87.779,Z 76.000,A 180.000,B 0.000,C 180.000} C_DIS
LIN {X 92.070,Y 87.864,Z 76.000,A 180.000,B 0.000,C 180.000} C_DIS
LIN {X 91.891,Y 87.969,Z 76.000,A 180.000,B 0.000,C 180.000} C_DIS
LIN {X 91.712,Y 88.075,Z 76.000,A 180.000,B 0.000,C 180.000} C_DIS
LIN {X 91.613,Y 88.137,Z 76.000,A 180.000,B 0.000,C 180.000} C_DIS
LIN {X 91.533,Y 88.187,Z 76.000,A 180.000,B 0.000,C 180.000} C_DIS
LIN {X 91.355,Y 88.307,Z 76.000,A 180.000,B 0.000,C 180.000} C_DIS
LIN {X 91.176,Y 88.426,Z 76.000,A 180.000,B 0.000,C 180.000} C_DIS
LIN {X 91.076,Y 88.494,Z 76.000,A 180.000,B 0.000,C 180.000} C_DIS
LIN {X 90.997,Y 88.553,Z 76.000,A 180.000,B 0.000,C 180.000} C_DIS
LIN {X 90.818,Y 88.688,Z 76.000,A 180.000,B 0.000,C 180.000} C_DIS
LIN {X 90.640,Y 88.823,Z 76.000,A 180.000,B 0.000,C 180.000} C_DIS
LIN {X 90.604,Y 88.852,Z 76.000,A 180.000,B 0.000,C 180.000} C_DIS
LIN {X 90.461,Y 88.971,Z 76.000,A 180.000,B 0.000,C 180.000} C_DIS
LIN {X 90.179,Y 89.209,Z 76.000,A 180.000,B 0.000,C 180.000} C_DIS
LIN {X 90.103,Y 89.275,Z 76.000,A 180.000,B 0.000,C 180.000} C_DIS
LIN {X 89.983,Y 89.388,Z 76.000,A 180.000,B 0.000,C 180.000} C_DIS
LIN {X 89.793,Y 89.567,Z 76.000,A 180.000,B 0.000,C 180.000} C_DIS
LIN {X 89.746,Y 89.612,Z 76.000,A 180.000,B 0.000,C 180.000} C_DIS
LIN {X 89.614,Y 89.746,Z 76.000,A 180.000,B 0.000,C 180.000} C_DIS
LIN {X 89.388,Y 89.985,Z 76.000,A 180.000,B 0.000,C 180.000} C_DIS
LIN {X 89.277,Y 90.103,Z 76.000,A 180.000,B 0.000,C 180.000} C_DIS
LIN {X 89.209,Y 90.177,Z 76.000,A 180.000,B 0.000,C 180.000} C_DIS
LIN {X 89.121,Y 90.282,Z 76.000,A 180.000,B 0.000,C 180.000} C_DIS
LIN {X 88.970,Y 90.461,Z 76.000,A 180.000,B 0.000,C 180.000} C_DIS
LIN {X 88.852,Y 90.603,Z 76.000,A 180.000,B 0.000,C 180.000} C_DIS
LIN {X 88.823,Y 90.640,Z 76.000,A 180.000,B 0.000,C 180.000} C_DIS
LIN {X 88.673,Y 90.839,Z 76.000,A 180.000,B 0.000,C 180.000} C_DIS
LIN {X 88.554,Y 90.997,Z 76.000,A 180.000,B 0.000,C 180.000} C_DIS
LIN {X 88.494,Y 91.080,Z 76.000,A 180.000,B 0.000,C 180.000} C_DIS
LIN {X 88.426,Y 91.176,Z 76.000,A 180.000,B 0.000,C 180.000} C_DIS
LIN {X 88.316,Y 91.340,Z 76.000,A 180.000,B 0.000,C 180.000} C_DIS
LIN {X 88.220,Y 91.484,Z 76.000,A 180.000,B 0.000,C 180.000} C_DIS
; Link Move Starts
LIN {X 88.064,Y 91.730,Z 76.000,A 180.000,B 0.000,C 180.000} C_DIS
LIN {X 87.907,Y 91.996,Z 75.999,A 180.000,B 0.000,C 180.000} C_DIS
LIN {X 87.760,Y 92.258,Z 75.998,A 180.000,B 0.000,C 180.000} C_DIS
LIN {X 87.619,Y 92.530,Z 75.996,A 180.000,B 0.000,C 180.000} C_DIS
LIN {X 87.485,Y 92.800,Z 75.994,A 180.000,B 0.000,C 180.000} C_DIS
LIN {X 87.360,Y 93.076,Z 75.992,A 180.000,B 0.000,C 180.000} C_DIS
LIN {X 87.246,Y 93.344,Z 75.989,A 180.000,B 0.000,C 180.000} C_DIS
LIN {X 87.132,Y 93.636,Z 75.986,A 180.000,B 0.000,C 180.000} C_DIS
LIN {X 87.028,Y 93.911,Z 75.983,A 180.000,B 0.000,C 180.000} C_DIS
LIN {X 86.932,Y 94.206,Z 75.978,A 180.000,B 0.000,C 180.000} C_DIS
LIN {X 86.845,Y 94.491,Z 75.974,A 180.000,B 0.000,C 180.000} C_DIS
LIN {X 86.766,Y 94.787,Z 75.969,A 180.000,B 0.000,C 180.000} C_DIS
LIN {X 86.691,Y 95.072,Z 75.964,A 180.000,B 0.000,C 180.000} C_DIS
LIN {X 86.659,Y 95.224,Z 75.962,A 180.000,B 0.000,C 180.000} C_DIS
LIN {X 86.627,Y 95.375,Z 75.959,A 180.000,B 0.000,C 180.000} C_DIS
LIN {X 86.597,Y 95.523,Z 75.956,A 180.000,B 0.000,C 180.000} C_DIS
LIN {X 86.569,Y 95.671,Z 75.953,A 180.000,B 0.000,C 180.000} C_DIS
LIN {X 86.546,Y 95.821,Z 75.950,A 180.000,B 0.000,C 180.000} C_DIS
LIN {X 86.523,Y 95.971,Z 75.947,A 180.000,B 0.000,C 180.000} C_DIS
LIN {X 86.501,Y 96.119,Z 75.944,A 180.000,B 0.000,C 180.000} C_DIS
LIN {X 86.480,Y 96.267,Z 75.940,A 180.000,B 0.000,C 180.000} C_DIS
LIN {X 86.464,Y 96.419,Z 75.937,A 180.000,B 0.000,C 180.000} C_DIS
LIN {X 86.449,Y 96.572,Z 75.934,A 180.000,B 0.000,C 180.000} C_DIS
LIN {X 86.435,Y 96.721,Z 75.930,A 180.000,B 0.000,C 180.000} C_DIS
LIN {X 86.422,Y 96.871,Z 75.926,A 180.000,B 0.000,C 180.000} C_DIS
LIN {X 86.415,Y 97.024,Z 75.923,A 180.000,B 0.000,C 180.000} C_DIS
LIN {X 86.409,Y 97.176,Z 75.919,A 180.000,B 0.000,C 180.000} C_DIS
LIN {X 86.403,Y 97.327,Z 75.915,A 180.000,B 0.000,C 180.000} C_DIS
LIN {X 86.399,Y 97.477,Z 75.911,A 180.000,B 0.000,C 180.000} C_DIS
LIN {X 86.398,Y 97.630,Z 75.907,A 180.000,B 0.000,C 180.000} C_DIS
LIN {X 86.400,Y 97.782,Z 75.903,A 180.000,B 0.000,C 180.000} C_DIS
LIN {X 86.402,Y 97.939,Z 75.899,A 180.000,B 0.000,C 180.000} C_DIS
LIN {X 86.405,Y 98.095,Z 75.895,A 180.000,B 0.000,C 180.000} C_DIS
LIN {X 86.413,Y 98.242,Z 75.890,A 180.000,B 0.000,C 180.000} C_DIS
LIN {X 86.424,Y 98.388,Z 75.886,A 180.000,B 0.000,C 180.000} C_DIS
LIN {X 86.434,Y 98.539,Z 75.882,A 180.000,B 0.000,C 180.000} C_DIS
LIN {X 86.446,Y 98.690,Z 75.877,A 180.000,B 0.000,C 180.000} C_DIS
LIN {X 86.462,Y 98.841,Z 75.873,A 180.000,B 0.000,C 180.000} C_DIS
LIN {X 86.481,Y 98.992,Z 75.868,A 180.000,B 0.000,C 180.000} C_DIS
LIN {X 86.501,Y 99.149,Z 75.863,A 180.000,B 0.000,C 180.000} C_DIS
LIN {X 86.521,Y 99.305,Z 75.858,A 180.000,B 0.000,C 180.000} C_DIS
LIN {X 86.543,Y 99.449,Z 75.854,A 180.000,B 0.000,C 180.000} C_DIS
LIN {X 86.569,Y 99.593,Z 75.849,A 180.000,B 0.000,C 180.000} C_DIS
LIN {X 86.597,Y 99.744,Z 75.844,A 180.000,B 0.000,C 180.000} C_DIS
LIN {X 86.624,Y 99.894,Z 75.839,A 180.000,B 0.000,C 180.000} C_DIS
LIN {X 86.639,Y 99.968,Z 75.837,A 180.000,B 0.000,C 180.000} C_DIS
LIN {X 86.657,Y 100.042,Z 75.834,A 180.000,B 0.000,C 180.000} C_DIS
LIN {X 86.674,Y 100.115,Z 75.832,A 180.000,B 0.000,C 180.000} C_DIS
LIN {X 86.692,Y 100.189,Z 75.829,A 180.000,B 0.000,C 180.000} C_DIS
LIN {X 86.711,Y 100.266,Z 75.826,A 180.000,B 0.000,C 180.000} C_DIS
LIN {X 86.729,Y 100.342,Z 75.824,A 180.000,B 0.000,C 180.000} C_DIS
LIN {X 86.748,Y 100.419,Z 75.821,A 180.000,B 0.000,C 180.000} C_DIS
LIN {X 86.766,Y 100.495,Z 75.818,A 180.000,B 0.000,C 180.000} C_DIS
LIN {X 86.783,Y 100.566,Z 75.816,A 180.000,B 0.000,C 180.000} C_DIS
LIN {X 86.802,Y 100.638,Z 75.813,A 180.000,B 0.000,C 180.000} C_DIS
LIN {X 86.823,Y 100.708,Z 75.811,A 180.000,B 0.000,C 180.000} C_DIS
LIN {X 86.844,Y 100.778,Z 75.808,A 180.000,B 0.000,C 180.000} C_DIS
LIN {X 86.888,Y 100.925,Z 75.803,A 180.000,B 0.000,C 180.000} C_DIS
LIN {X 86.932,Y 101.071,Z 75.797,A 180.000,B 0.000,C 180.000} C_DIS
LIN {X 86.954,Y 101.144,Z 75.795,A 180.000,B 0.000,C 180.000} C_DIS
LIN {X 86.979,Y 101.216,Z 75.792,A 180.000,B 0.000,C 180.000} C_DIS
LIN {X 87.005,Y 101.287,Z 75.790,A 180.000,B 0.000,C 180.000} C_DIS
LIN {X 87.030,Y 101.358,Z 75.787,A 180.000,B 0.000,C 180.000} C_DIS
LIN {X 87.084,Y 101.505,Z 75.781,A 180.000,B 0.000,C 180.000} C_DIS
LIN {X 87.110,Y 101.578,Z 75.779,A 180.000,B 0.000,C 180.000} C_DIS
LIN {X 87.137,Y 101.652,Z 75.776,A 180.000,B 0.000,C 180.000} C_DIS
LIN {X 87.163,Y 101.722,Z 75.773,A 180.000,B 0.000,C 180.000} C_DIS
LIN {X 87.190,Y 101.791,Z 75.771,A 180.000,B 0.000,C 180.000} C_DIS
LIN {X 87.217,Y 101.860,Z 75.768,A 180.000,B 0.000,C 180.000} C_DIS
LIN {X 87.247,Y 101.929,Z 75.766,A 180.000,B 0.000,C 180.000} C_DIS
LIN {X 87.308,Y 102.073,Z 75.760,A 180.000,B 0.000,C 180.000} C_DIS
LIN {X 87.370,Y 102.218,Z 75.755,A 180.000,B 0.000,C 180.000} C_DIS
LIN {X 87.399,Y 102.286,Z 75.752,A 180.000,B 0.000,C 180.000} C_DIS
LIN {X 87.430,Y 102.353,Z 75.749,A 180.000,B 0.000,C 180.000} C_DIS
LIN {X 87.462,Y 102.420,Z 75.747,A 180.000,B 0.000,C 180.000} C_DIS
LIN {X 87.495,Y 102.486,Z 75.744,A 180.000,B 0.000,C 180.000} C_DIS
LIN {X 87.565,Y 102.627,Z 75.739,A 180.000,B 0.000,C 180.000} C_DIS
LIN {X 87.635,Y 102.768,Z 75.733,A 180.000,B 0.000,C 180.000} C_DIS
LIN {X 87.668,Y 102.834,Z 75.731,A 180.000,B 0.000,C 180.000} C_DIS
LIN {X 87.703,Y 102.900,Z 75.728,A 180.000,B 0.000,C 180.000} C_DIS
LIN {X 87.737,Y 102.965,Z 75.726,A 180.000,B 0.000,C 180.000} C_DIS
LIN {X 87.773,Y 103.030,Z 75.723,A 180.000,B 0.000,C 180.000} C_DIS
LIN {X 87.851,Y 103.167,Z 75.717,A 180.000,B 0.000,C 180.000} C_DIS
LIN {X 87.965,Y 103.368,Z 75.709,A 180.000,B 0.000,C 180.000} C_DIS
LIN {X 88.002,Y 103.433,Z 75.707,A 180.000,B 0.000,C 180.000} C_DIS
LIN {X 88.041,Y 103.496,Z 75.704,A 180.000,B 0.000,C 180.000} C_DIS
LIN {X 88.081,Y 103.559,Z 75.702,A 180.000,B 0.000,C 180.000} C_DIS
LIN {X 88.166,Y 103.691,Z 75.696,A 180.000,B 0.000,C 180.000} C_DIS
LIN {X 88.292,Y 103.886,Z 75.688,A 180.000,B 0.000,C 180.000} C_DIS
LIN {X 88.333,Y 103.948,Z 75.685,A 180.000,B 0.000,C 180.000} C_DIS
LIN {X 88.376,Y 104.009,Z 75.683,A 180.000,B 0.000,C 180.000} C_DIS
LIN {X 88.419,Y 104.070,Z 75.680,A 180.000,B 0.000,C 180.000} C_DIS
LIN {X 88.465,Y 104.134,Z 75.677,A 180.000,B 0.000,C 180.000} C_DIS
LIN {X 88.557,Y 104.261,Z 75.672,A 180.000,B 0.000,C 180.000} C_DIS
LIN {X 88.603,Y 104.324,Z 75.669,A 180.000,B 0.000,C 180.000} C_DIS
LIN {X 88.692,Y 104.446,Z 75.664,A 180.000,B 0.000,C 180.000} C_DIS
LIN {X 88.737,Y 104.506,Z 75.661,A 180.000,B 0.000,C 180.000} C_DIS
LIN {X 88.783,Y 104.565,Z 75.659,A 180.000,B 0.000,C 180.000} C_DIS
LIN {X 88.931,Y 104.746,Z 75.651,A 180.000,B 0.000,C 180.000} C_DIS
LIN {X 89.028,Y 104.865,Z 75.645,A 180.000,B 0.000,C 180.000} C_DIS
LIN {X 89.076,Y 104.923,Z 75.643,A 180.000,B 0.000,C 180.000} C_DIS
LIN {X 89.126,Y 104.981,Z 75.640,A 180.000,B 0.000,C 180.000} C_DIS
LIN {X 89.176,Y 105.037,Z 75.637,A 180.000,B 0.000,C 180.000} C_DIS
LIN {X 89.229,Y 105.094,Z 75.635,A 180.000,B 0.000,C 180.000} C_DIS
LIN {X 89.487,Y 105.377,Z 75.621,A 180.000,B 0.000,C 180.000} C_DIS
LIN {X 89.538,Y 105.432,Z 75.619,A 180.000,B 0.000,C 180.000} C_DIS
LIN {X 89.590,Y 105.486,Z 75.616,A 180.000,B 0.000,C 180.000} C_DIS
LIN {X 89.646,Y 105.542,Z 75.613,A 180.000,B 0.000,C 180.000} C_DIS
LIN {X 89.923,Y 105.813,Z 75.600,A 180.000,B 0.000,C 180.000} C_DIS
LIN {X 89.978,Y 105.865,Z 75.597,A 180.000,B 0.000,C 180.000} C_DIS
LIN {X 90.035,Y 105.916,Z 75.594,A 180.000,B 0.000,C 180.000} C_DIS
LIN {X 90.210,Y 106.069,Z 75.586,A 180.000,B 0.000,C 180.000} C_DIS
LIN {X 90.327,Y 106.171,Z 75.581,A 180.000,B 0.000,C 180.000} C_DIS
LIN {X 90.385,Y 106.222,Z 75.578,A 180.000,B 0.000,C 180.000} C_DIS
LIN {X 90.444,Y 106.272,Z 75.575,A 180.000,B 0.000,C 180.000} C_DIS
LIN {X 90.503,Y 106.323,Z 75.573,A 180.000,B 0.000,C 180.000} C_DIS
LIN {X 90.562,Y 106.371,Z 75.570,A 180.000,B 0.000,C 180.000} C_DIS
LIN {X 90.743,Y 106.511,Z 75.562,A 180.000,B 0.000,C 180.000} C_DIS
LIN {X 90.863,Y 106.604,Z 75.557,A 180.000,B 0.000,C 180.000} C_DIS
LIN {X 90.923,Y 106.651,Z 75.554,A 180.000,B 0.000,C 180.000} C_DIS
LIN {X 90.983,Y 106.696,Z 75.551,A 180.000,B 0.000,C 180.000} C_DIS
LIN {X 91.047,Y 106.741,Z 75.549,A 180.000,B 0.000,C 180.000} C_DIS
LIN {X 91.367,Y 106.962,Z 75.535,A 180.000,B 0.000,C 180.000} C_DIS
LIN {X 91.431,Y 107.006,Z 75.532,A 180.000,B 0.000,C 180.000} C_DIS
LIN {X 91.495,Y 107.048,Z 75.530,A 180.000,B 0.000,C 180.000} C_DIS
LIN {X 91.560,Y 107.090,Z 75.527,A 180.000,B 0.000,C 180.000} C_DIS
LIN {X 91.625,Y 107.131,Z 75.524,A 180.000,B 0.000,C 180.000} C_DIS
LIN {X 91.952,Y 107.331,Z 75.511,A 180.000,B 0.000,C 180.000} C_DIS
LIN {X 92.018,Y 107.371,Z 75.508,A 180.000,B 0.000,C 180.000} C_DIS
LIN {X 92.085,Y 107.409,Z 75.506,A 180.000,B 0.000,C 180.000} C_DIS
LIN {X 92.153,Y 107.446,Z 75.503,A 180.000,B 0.000,C 180.000} C_DIS
LIN {X 92.493,Y 107.628,Z 75.489,A 180.000,B 0.000,C 180.000} C_DIS
LIN {X 92.561,Y 107.663,Z 75.487,A 180.000,B 0.000,C 180.000} C_DIS
LIN {X 92.631,Y 107.698,Z 75.484,A 180.000,B 0.000,C 180.000} C_DIS
LIN {X 92.700,Y 107.732,Z 75.481,A 180.000,B 0.000,C 180.000} C_DIS
LIN {X 92.770,Y 107.765,Z 75.479,A 180.000,B 0.000,C 180.000} C_DIS
LIN {X 93.125,Y 107.930,Z 75.465,A 180.000,B 0.000,C 180.000} C_DIS
LIN {X 93.194,Y 107.961,Z 75.462,A 180.000,B 0.000,C 180.000} C_DIS
LIN {X 93.265,Y 107.990,Z 75.460,A 180.000,B 0.000,C 180.000} C_DIS
LIN {X 93.623,Y 108.134,Z 75.446,A 180.000,B 0.000,C 180.000} C_DIS
LIN {X 93.696,Y 108.162,Z 75.443,A 180.000,B 0.000,C 180.000} C_DIS
LIN {X 93.768,Y 108.189,Z 75.441,A 180.000,B 0.000,C 180.000} C_DIS
LIN {X 93.840,Y 108.214,Z 75.438,A 180.000,B 0.000,C 180.000} C_DIS
LIN {X 93.913,Y 108.238,Z 75.435,A 180.000,B 0.000,C 180.000} C_DIS
LIN {X 94.280,Y 108.362,Z 75.422,A 180.000,B 0.000,C 180.000} C_DIS
LIN {X 94.353,Y 108.387,Z 75.419,A 180.000,B 0.000,C 180.000} C_DIS
LIN {X 94.427,Y 108.409,Z 75.416,A 180.000,B 0.000,C 180.000} C_DIS
LIN {X 94.501,Y 108.430,Z 75.414,A 180.000,B 0.000,C 180.000} C_DIS
LIN {X 94.726,Y 108.492,Z 75.406,A 180.000,B 0.000,C 180.000} C_DIS
LIN {X 94.878,Y 108.533,Z 75.400,A 180.000,B 0.000,C 180.000} C_DIS
LIN {X 94.952,Y 108.553,Z 75.397,A 180.000,B 0.000,C 180.000} C_DIS
LIN {X 95.026,Y 108.570,Z 75.395,A 180.000,B 0.000,C 180.000} C_DIS
LIN {X 95.407,Y 108.652,Z 75.381,A 180.000,B 0.000,C 180.000} C_DIS
LIN {X 95.484,Y 108.668,Z 75.378,A 180.000,B 0.000,C 180.000} C_DIS
LIN {X 95.559,Y 108.684,Z 75.376,A 180.000,B 0.000,C 180.000} C_DIS
LIN {X 95.633,Y 108.699,Z 75.373,A 180.000,B 0.000,C 180.000} C_DIS
LIN {X 95.709,Y 108.712,Z 75.370,A 180.000,B 0.000,C 180.000} C_DIS
LIN {X 95.862,Y 108.736,Z 75.365,A 180.000,B 0.000,C 180.000} C_DIS
LIN {X 96.095,Y 108.773,Z 75.357,A 180.000,B 0.000,C 180.000} C_DIS
LIN {X 96.170,Y 108.785,Z 75.354,A 180.000,B 0.000,C 180.000} C_DIS
LIN {X 96.246,Y 108.795,Z 75.351,A 180.000,B 0.000,C 180.000} C_DIS
LIN {X 96.322,Y 108.803,Z 75.349,A 180.000,B 0.000,C 180.000} C_DIS
LIN {X 96.399,Y 108.810,Z 75.346,A 180.000,B 0.000,C 180.000} C_DIS
LIN {X 96.555,Y 108.826,Z 75.341,A 180.000,B 0.000,C 180.000} C_DIS
LIN {X 96.712,Y 108.842,Z 75.335,A 180.000,B 0.000,C 180.000} C_DIS
LIN {X 96.789,Y 108.849,Z 75.332,A 180.000,B 0.000,C 180.000} C_DIS
LIN {X 96.865,Y 108.855,Z 75.330,A 180.000,B 0.000,C 180.000} C_DIS
LIN {X 96.942,Y 108.861,Z 75.327,A 180.000,B 0.000,C 180.000} C_DIS
LIN {X 97.019,Y 108.865,Z 75.324,A 180.000,B 0.000,C 180.000} C_DIS
LIN {X 97.176,Y 108.871,Z 75.319,A 180.000,B 0.000,C 180.000} C_DIS
LIN {X 97.409,Y 108.882,Z 75.311,A 180.000,B 0.000,C 180.000} C_DIS
LIN {X 97.486,Y 108.885,Z 75.308,A 180.000,B 0.000,C 180.000} C_DIS
LIN {X 97.563,Y 108.885,Z 75.305,A 180.000,B 0.000,C 180.000} C_DIS
LIN {X 97.639,Y 108.884,Z 75.303,A 180.000,B 0.000,C 180.000} C_DIS
LIN {X 97.797,Y 108.882,Z 75.297,A 180.000,B 0.000,C 180.000} C_DIS
LIN {X 97.954,Y 108.881,Z 75.292,A 180.000,B 0.000,C 180.000} C_DIS
LIN {X 98.032,Y 108.880,Z 75.289,A 180.000,B 0.000,C 180.000} C_DIS
LIN {X 98.109,Y 108.877,Z 75.286,A 180.000,B 0.000,C 180.000} C_DIS
LIN {X 98.186,Y 108.873,Z 75.284,A 180.000,B 0.000,C 180.000} C_DIS
LIN {X 98.263,Y 108.869,Z 75.281,A 180.000,B 0.000,C 180.000} C_DIS
LIN {X 98.341,Y 108.864,Z 75.278,A 180.000,B 0.000,C 180.000} C_DIS
LIN {X 98.498,Y 108.854,Z 75.273,A 180.000,B 0.000,C 180.000} C_DIS
LIN {X 98.576,Y 108.848,Z 75.270,A 180.000,B 0.000,C 180.000} C_DIS
LIN {X 98.653,Y 108.843,Z 75.267,A 180.000,B 0.000,C 180.000} C_DIS
LIN {X 98.730,Y 108.838,Z 75.265,A 180.000,B 0.000,C 180.000} C_DIS
LIN {X 98.807,Y 108.831,Z 75.262,A 180.000,B 0.000,C 180.000} C_DIS
LIN {X 98.883,Y 108.822,Z 75.259,A 180.000,B 0.000,C 180.000} C_DIS
LIN {X 99.039,Y 108.803,Z 75.254,A 180.000,B 0.000,C 180.000} C_DIS
LIN {X 99.273,Y 108.774,Z 75.245,A 180.000,B 0.000,C 180.000} C_DIS
LIN {X 99.349,Y 108.764,Z 75.243,A 180.000,B 0.000,C 180.000} C_DIS
LIN {X 99.426,Y 108.751,Z 75.240,A 180.000,B 0.000,C 180.000} C_DIS
LIN {X 99.502,Y 108.738,Z 75.237,A 180.000,B 0.000,C 180.000} C_DIS
LIN {X 99.579,Y 108.724,Z 75.235,A 180.000,B 0.000,C 180.000} C_DIS
LIN {X 99.734,Y 108.696,Z 75.229,A 180.000,B 0.000,C 180.000} C_DIS
LIN {X 99.811,Y 108.682,Z 75.226,A 180.000,B 0.000,C 180.000} C_DIS
LIN {X 99.963,Y 108.655,Z 75.221,A 180.000,B 0.000,C 180.000} C_DIS
LIN {X 100.039,Y 108.640,Z 75.218,A 180.000,B 0.000,C 180.000} C_DIS
LIN {X 100.115,Y 108.624,Z 75.216,A 180.000,B 0.000,C 180.000} C_DIS
LIN {X 100.192,Y 108.606,Z 75.213,A 180.000,B 0.000,C 180.000} C_DIS
LIN {X 100.345,Y 108.569,Z 75.207,A 180.000,B 0.000,C 180.000} C_DIS
LIN {X 100.421,Y 108.550,Z 75.205,A 180.000,B 0.000,C 180.000} C_DIS
LIN {X 100.572,Y 108.514,Z 75.199,A 180.000,B 0.000,C 180.000} C_DIS
LIN {X 100.647,Y 108.495,Z 75.196,A 180.000,B 0.000,C 180.000} C_DIS
LIN {X 100.722,Y 108.473,Z 75.194,A 180.000,B 0.000,C 180.000} C_DIS
LIN {X 100.872,Y 108.428,Z 75.188,A 180.000,B 0.000,C 180.000} C_DIS
LIN {X 100.948,Y 108.405,Z 75.186,A 180.000,B 0.000,C 180.000} C_DIS
LIN {X 101.023,Y 108.382,Z 75.183,A 180.000,B 0.000,C 180.000} C_DIS
LIN {X 101.098,Y 108.360,Z 75.180,A 180.000,B 0.000,C 180.000} C_DIS
LIN {X 101.173,Y 108.337,Z 75.177,A 180.000,B 0.000,C 180.000} C_DIS
LIN {X 101.248,Y 108.314,Z 75.175,A 180.000,B 0.000,C 180.000} C_DIS
LIN {X 101.323,Y 108.290,Z 75.172,A 180.000,B 0.000,C 180.000} C_DIS
LIN {X 101.397,Y 108.264,Z 75.170,A 180.000,B 0.000,C 180.000} C_DIS
LIN {X 101.470,Y 108.238,Z 75.167,A 180.000,B 0.000,C 180.000} C_DIS
LIN {X 101.543,Y 108.211,Z 75.164,A 180.000,B 0.000,C 180.000} C_DIS
LIN {X 101.616,Y 108.184,Z 75.162,A 180.000,B 0.000,C 180.000} C_DIS
LIN {X 101.689,Y 108.158,Z 75.159,A 180.000,B 0.000,C 180.000} C_DIS
LIN {X 101.762,Y 108.131,Z 75.157,A 180.000,B 0.000,C 180.000} C_DIS
LIN {X 101.908,Y 108.075,Z 75.152,A 180.000,B 0.000,C 180.000} C_DIS
LIN {X 101.980,Y 108.044,Z 75.149,A 180.000,B 0.000,C 180.000} C_DIS
LIN {X 102.052,Y 108.013,Z 75.147,A 180.000,B 0.000,C 180.000} C_DIS
LIN {X 102.197,Y 107.951,Z 75.142,A 180.000,B 0.000,C 180.000} C_DIS
LIN {X 102.341,Y 107.889,Z 75.137,A 180.000,B 0.000,C 180.000} C_DIS
LIN {X 102.484,Y 107.825,Z 75.132,A 180.000,B 0.000,C 180.000} C_DIS
LIN {X 102.625,Y 107.757,Z 75.128,A 180.000,B 0.000,C 180.000} C_DIS
LIN {X 102.765,Y 107.687,Z 75.123,A 180.000,B 0.000,C 180.000} C_DIS
LIN {X 102.905,Y 107.617,Z 75.118,A 180.000,B 0.000,C 180.000} C_DIS
LIN {X 103.045,Y 107.547,Z 75.114,A 180.000,B 0.000,C 180.000} C_DIS
LIN {X 103.182,Y 107.470,Z 75.109,A 180.000,B 0.000,C 180.000} C_DIS
LIN {X 103.318,Y 107.392,Z 75.105,A 180.000,B 0.000,C 180.000} C_DIS
LIN {X 103.454,Y 107.314,Z 75.101,A 180.000,B 0.000,C 180.000} C_DIS
LIN {X 103.590,Y 107.234,Z 75.096,A 180.000,B 0.000,C 180.000} C_DIS
LIN {X 103.722,Y 107.151,Z 75.092,A 180.000,B 0.000,C 180.000} C_DIS
LIN {X 103.854,Y 107.065,Z 75.088,A 180.000,B 0.000,C 180.000} C_DIS
LIN {X 103.986,Y 106.980,Z 75.084,A 180.000,B 0.000,C 180.000} C_DIS
LIN {X 104.118,Y 106.894,Z 75.080,A 180.000,B 0.000,C 180.000} C_DIS
LIN {X 104.245,Y 106.803,Z 75.076,A 180.000,B 0.000,C 180.000} C_DIS
LIN {X 104.372,Y 106.710,Z 75.073,A 180.000,B 0.000,C 180.000} C_DIS
LIN {X 104.498,Y 106.617,Z 75.069,A 180.000,B 0.000,C 180.000} C_DIS
LIN {X 104.624,Y 106.524,Z 75.065,A 180.000,B 0.000,C 180.000} C_DIS
LIN {X 104.747,Y 106.426,Z 75.062,A 180.000,B 0.000,C 180.000} C_DIS
LIN {X 104.868,Y 106.326,Z 75.058,A 180.000,B 0.000,C 180.000} C_DIS
LIN {X 104.989,Y 106.225,Z 75.055,A 180.000,B 0.000,C 180.000} C_DIS
LIN {X 105.110,Y 106.125,Z 75.052,A 180.000,B 0.000,C 180.000} C_DIS
LIN {X 105.229,Y 106.022,Z 75.049,A 180.000,B 0.000,C 180.000} C_DIS
LIN {X 105.344,Y 105.915,Z 75.045,A 180.000,B 0.000,C 180.000} C_DIS
LIN {X 105.460,Y 105.808,Z 75.042,A 180.000,B 0.000,C 180.000} C_DIS
LIN {X 105.575,Y 105.701,Z 75.040,A 180.000,B 0.000,C 180.000} C_DIS
LIN {X 105.686,Y 105.590,Z 75.037,A 180.000,B 0.000,C 180.000} C_DIS
LIN {X 105.795,Y 105.477,Z 75.034,A 180.000,B 0.000,C 180.000} C_DIS
LIN {X 105.904,Y 105.363,Z 75.031,A 180.000,B 0.000,C 180.000} C_DIS
LIN {X 106.013,Y 105.250,Z 75.029,A 180.000,B 0.000,C 180.000} C_DIS
LIN {X 106.223,Y 105.016,Z 75.024,A 180.000,B 0.000,C 180.000} C_DIS
LIN {X 106.428,Y 104.776,Z 75.020,A 180.000,B 0.000,C 180.000} C_DIS
LIN {X 106.623,Y 104.530,Z 75.016,A 180.000,B 0.000,C 180.000} C_DIS
LIN {X 106.814,Y 104.279,Z 75.012,A 180.000,B 0.000,C 180.000} C_DIS
LIN {X 106.997,Y 104.023,Z 75.009,A 180.000,B 0.000,C 180.000} C_DIS
LIN {X 107.173,Y 103.762,Z 75.006,A 180.000,B 0.000,C 180.000} C_DIS
LIN {X 107.341,Y 103.496,Z 75.004,A 180.000,B 0.000,C 180.000} C_DIS
LIN {X 107.502,Y 103.225,Z 75.002,A 180.000,B 0.000,C 180.000} C_DIS
LIN {X 107.655,Y 102.950,Z 75.001,A 180.000,B 0.000,C 180.000} C_DIS
LIN {X 107.800,Y 102.670,Z 75.000,A 180.000,B 0.000,C 180.000} C_DIS
LIN {X 107.939,Y 102.388,Z 75.000,A 180.000,B 0.000,C 180.000} C_DIS
LIN {X 107.965,Y 102.330,Z 75.000,A 180.000,B 0.000,C 180.000} C_DIS
; Cutting Move Starts
LIN {X 107.996,Y 102.260,Z 75.000,A 180.000,B 0.000,C 180.000} C_DIS
LIN {X 108.076,Y 102.081,Z 75.000,A 180.000,B 0.000,C 180.000} C_DIS
LIN {X 108.153,Y 101.902,Z 75.000,A 180.000,B 0.000,C 180.000} C_DIS
LIN {X 108.159,Y 101.887,Z 75.000,A 180.000,B 0.000,C 180.000} C_DIS
LIN {X 108.223,Y 101.723,Z 75.000,A 180.000,B 0.000,C 180.000} C_DIS
LIN {X 108.359,Y 101.366,Z 75.000,A 180.000,B 0.000,C 180.000} C_DIS
LIN {X 108.421,Y 101.187,Z 75.000,A 180.000,B 0.000,C 180.000} C_DIS
LIN {X 108.535,Y 100.829,Z 75.000,A 180.000,B 0.000,C 180.000} C_DIS
LIN {X 108.588,Y 100.651,Z 75.000,A 180.000,B 0.000,C 180.000} C_DIS
LIN {X 108.695,Y 100.234,Z 75.000,A 180.000,B 0.000,C 180.000} C_DIS
LIN {X 108.726,Y 100.114,Z 75.000,A 180.000,B 0.000,C 180.000} C_DIS
LIN {X 108.766,Y 99.936,Z 75.000,A 180.000,B 0.000,C 180.000} C_DIS
LIN {X 108.838,Y 99.578,Z 75.000,A 180.000,B 0.000,C 180.000} C_DIS
LIN {X 108.870,Y 99.399,Z 75.000,A 180.000,B 0.000,C 180.000} C_DIS
LIN {X 108.874,Y 99.372,Z 75.000,A 180.000,B 0.000,C 180.000} C_DIS
LIN {X 108.921,Y 99.042,Z 75.000,A 180.000,B 0.000,C 180.000} C_DIS
LIN {X 108.945,Y 98.863,Z 75.000,A 180.000,B 0.000,C 180.000} C_DIS
LIN {X 108.966,Y 98.684,Z 75.000,A 180.000,B 0.000,C 180.000} C_DIS
LIN {X 108.996,Y 98.327,Z 75.000,A 180.000,B 0.000,C 180.000} C_DIS
LIN {X 109.010,Y 98.148,Z 75.000,A 180.000,B 0.000,C 180.000} C_DIS
LIN {X 109.016,Y 97.969,Z 75.000,A 180.000,B 0.000,C 180.000} C_DIS
LIN {X 109.021,Y 97.790,Z 75.000,A 180.000,B 0.000,C 180.000} C_DIS
LIN {X 109.026,Y 97.612,Z 75.000,A 180.000,B 0.000,C 180.000} C_DIS
LIN {X 109.027,Y 97.433,Z 75.000,A 180.000,B 0.000,C 180.000} C_DIS
LIN {X 109.022,Y 97.254,Z 75.000,A 180.000,B 0.000,C 180.000} C_DIS
LIN {X 109.017,Y 97.075,Z 75.000,A 180.000,B 0.000,C 180.000} C_DIS
LIN {X 109.012,Y 96.897,Z 75.000,A 180.000,B 0.000,C 180.000} C_DIS
LIN {X 109.000,Y 96.718,Z 75.000,A 180.000,B 0.000,C 180.000} C_DIS
LIN {X 108.970,Y 96.360,Z 75.000,A 180.000,B 0.000,C 180.000} C_DIS
LIN {X 108.951,Y 96.181,Z 75.000,A 180.000,B 0.000,C 180.000} C_DIS
LIN {X 108.927,Y 96.003,Z 75.000,A 180.000,B 0.000,C 180.000} C_DIS
LIN {X 108.874,Y 95.628,Z 75.000,A 180.000,B 0.000,C 180.000} C_DIS
LIN {X 108.846,Y 95.466,Z 75.000,A 180.000,B 0.000,C 180.000} C_DIS
LIN {X 108.775,Y 95.109,Z 75.000,A 180.000,B 0.000,C 180.000} C_DIS
LIN {X 108.737,Y 94.930,Z 75.000,A 180.000,B 0.000,C 180.000} C_DIS
LIN {X 108.695,Y 94.766,Z 75.000,A 180.000,B 0.000,C 180.000} C_DIS
LIN {X 108.599,Y 94.394,Z 75.000,A 180.000,B 0.000,C 180.000} C_DIS
LIN {X 108.549,Y 94.215,Z 75.000,A 180.000,B 0.000,C 180.000} C_DIS
LIN {X 108.435,Y 93.857,Z 75.000,A 180.000,B 0.000,C 180.000} C_DIS
LIN {X 108.376,Y 93.679,Z 75.000,A 180.000,B 0.000,C 180.000} C_DIS
LIN {X 108.338,Y 93.578,Z 75.000,A 180.000,B 0.000,C 180.000} C_DIS
LIN {X 108.240,Y 93.321,Z 75.000,A 180.000,B 0.000,C 180.000} C_DIS
LIN {X 108.171,Y 93.142,Z 75.000,A 180.000,B 0.000,C 180.000} C_DIS
LIN {X 108.159,Y 93.113,Z 75.000,A 180.000,B 0.000,C 180.000} C_DIS
LIN {X 108.096,Y 92.964,Z 75.000,A 180.000,B 0.000,C 180.000} C_DIS
LIN {X 107.936,Y 92.606,Z 75.000,A 180.000,B 0.000,C 180.000} C_DIS
LIN {X 107.851,Y 92.427,Z 75.000,A 180.000,B 0.000,C 180.000} C_DIS
LIN {X 107.666,Y 92.070,Z 75.000,A 180.000,B 0.000,C 180.000} C_DIS
LIN {X 107.623,Y 91.987,Z 75.000,A 180.000,B 0.000,C 180.000} C_DIS
LIN {X 107.570,Y 91.891,Z 75.000,A 180.000,B 0.000,C 180.000} C_DIS
LIN {X 107.466,Y 91.712,Z 75.000,A 180.000,B 0.000,C 180.000} C_DIS
LIN {X 107.361,Y 91.533,Z 75.000,A 180.000,B 0.000,C 180.000} C_DIS
LIN {X 107.265,Y 91.373,Z 75.000,A 180.000,B 0.000,C 180.000} C_DIS
LIN {X 107.254,Y 91.355,Z 75.000,A 180.000,B 0.000,C 180.000} C_DIS
LIN {X 107.135,Y 91.176,Z 75.000,A 180.000,B 0.000,C 180.000} C_DIS
LIN {X 107.016,Y 90.997,Z 75.000,A 180.000,B 0.000,C 180.000} C_DIS
LIN {X 106.908,Y 90.839,Z 75.000,A 180.000,B 0.000,C 180.000} C_DIS
LIN {X 106.893,Y 90.818,Z 75.000,A 180.000,B 0.000,C 180.000} C_DIS
LIN {X 106.760,Y 90.640,Z 75.000,A 180.000,B 0.000,C 180.000} C_DIS
LIN {X 106.550,Y 90.361,Z 75.000,A 180.000,B 0.000,C 180.000} C_DIS
LIN {X 106.489,Y 90.282,Z 75.000,A 180.000,B 0.000,C 180.000} C_DIS
LIN {X 106.371,Y 90.142,Z 75.000,A 180.000,B 0.000,C 180.000} C_DIS
LIN {X 106.187,Y 89.925,Z 75.000,A 180.000,B 0.000,C 180.000} C_DIS
LIN {X 106.027,Y 89.746,Z 75.000,A 180.000,B 0.000,C 180.000} C_DIS
LIN {X 106.014,Y 89.732,Z 75.000,A 180.000,B 0.000,C 180.000} C_DIS
LIN {X 105.858,Y 89.567,Z 75.000,A 180.000,B 0.000,C 180.000} C_DIS
LIN {X 105.689,Y 89.388,Z 75.000,A 180.000,B 0.000,C 180.000} C_DIS
LIN {X 105.656,Y 89.354,Z 75.000,A 180.000,B 0.000,C 180.000} C_DIS
LIN {X 105.507,Y 89.209,Z 75.000,A 180.000,B 0.000,C 180.000} C_DIS
LIN {X 105.299,Y 89.013,Z 75.000,A 180.000,B 0.000,C 180.000} C_DIS
LIN {X 105.120,Y 88.852,Z 75.000,A 180.000,B 0.000,C 180.000} C_DIS
LIN {X 104.909,Y 88.673,Z 75.000,A 180.000,B 0.000,C 180.000} C_DIS
LIN {X 104.762,Y 88.550,Z 75.000,A 180.000,B 0.000,C 180.000} C_DIS
LIN {X 104.695,Y 88.494,Z 75.000,A 180.000,B 0.000,C 180.000} C_DIS
LIN {X 104.584,Y 88.407,Z 75.000,A 180.000,B 0.000,C 180.000} C_DIS
LIN {X 104.405,Y 88.272,Z 75.000,A 180.000,B 0.000,C 180.000} C_DIS
LIN {X 104.226,Y 88.138,Z 75.000,A 180.000,B 0.000,C 180.000} C_DIS
LIN {X 104.225,Y 88.137,Z 75.000,A 180.000,B 0.000,C 180.000} C_DIS
LIN {X 104.047,Y 88.014,Z 75.000,A 180.000,B 0.000,C 180.000} C_DIS
LIN {X 103.869,Y 87.895,Z 75.000,A 180.000,B 0.000,C 180.000} C_DIS
LIN {X 103.694,Y 87.779,Z 75.000,A 180.000,B 0.000,C 180.000} C_DIS
LIN {X 103.690,Y 87.776,Z 75.000,A 180.000,B 0.000,C 180.000} C_DIS
LIN {X 103.511,Y 87.665,Z 75.000,A 180.000,B 0.000,C 180.000} C_DIS
LIN {X 103.153,Y 87.455,Z 75.000,A 180.000,B 0.000,C 180.000} C_DIS
LIN {X 103.097,Y 87.422,Z 75.000,A 180.000,B 0.000,C 180.000} C_DIS
LIN {X 102.975,Y 87.356,Z 75.000,A 180.000,B 0.000,C 180.000} C_DIS
LIN {X 102.617,Y 87.172,Z 75.000,A 180.000,B 0.000,C 180.000} C_DIS
LIN {X 102.438,Y 87.085,Z 75.000,A 180.000,B 0.000,C 180.000} C_DIS
LIN {X 102.393,Y 87.064,Z 75.000,A 180.000,B 0.000,C 180.000} C_DIS
LIN {X 102.260,Y 87.004,Z 75.000,A 180.000,B 0.000,C 180.000} C_DIS
LIN {X 101.994,Y 86.885,Z 75.000,A 180.000,B 0.000,C 180.000} C_DIS
LIN {X 101.902,Y 86.845,Z 75.000,A 180.000,B 0.000,C 180.000} C_DIS
LIN {X 101.723,Y 86.776,Z 75.000,A 180.000,B 0.000,C 180.000} C_DIS
LIN {X 101.542,Y 86.707,Z 75.000,A 180.000,B 0.000,C 180.000} C_DIS
LIN {X 101.366,Y 86.640,Z 75.000,A 180.000,B 0.000,C 180.000} C_DIS
LIN {X 101.187,Y 86.580,Z 75.000,A 180.000,B 0.000,C 180.000} C_DIS
LIN {X 101.008,Y 86.523,Z 75.000,A 180.000,B 0.000,C 180.000} C_DIS
LIN {X 100.829,Y 86.466,Z 75.000,A 180.000,B 0.000,C 180.000} C_DIS
LIN {X 100.651,Y 86.411,Z 75.000,A 180.000,B 0.000,C 180.000} C_DIS
LIN {X 100.472,Y 86.364,Z 75.000,A 180.000,B 0.000,C 180.000} C_DIS
LIN {X 100.293,Y 86.318,Z 75.000,A 180.000,B 0.000,C 180.000} C_DIS
LIN {X 100.114,Y 86.272,Z 75.000,A 180.000,B 0.000,C 180.000} C_DIS
LIN {X 99.936,Y 86.235,Z 75.000,A 180.000,B 0.000,C 180.000} C_DIS
LIN {X 99.578,Y 86.164,Z 75.000,A 180.000,B 0.000,C 180.000} C_DIS
LIN {X 99.399,Y 86.130,Z 75.000,A 180.000,B 0.000,C 180.000} C_DIS
LIN {X 99.221,Y 86.104,Z 75.000,A 180.000,B 0.000,C 180.000} C_DIS
LIN {X 99.042,Y 86.078,Z 75.000,A 180.000,B 0.000,C 180.000} C_DIS
LIN {X 98.863,Y 86.053,Z 75.000,A 180.000,B 0.000,C 180.000} C_DIS
LIN {X 98.684,Y 86.035,Z 75.000,A 180.000,B 0.000,C 180.000} C_DIS
LIN {X 98.327,Y 86.004,Z 75.000,A 180.000,B 0.000,C 180.000} C_DIS
LIN {X 98.148,Y 85.992,Z 75.000,A 180.000,B 0.000,C 180.000} C_DIS
LIN {X 97.969,Y 85.984,Z 75.000,A 180.000,B 0.000,C 180.000} C_DIS
LIN {X 97.612,Y 85.974,Z 75.000,A 180.000,B 0.000,C 180.000} C_DIS
LIN {X 97.433,Y 85.973,Z 75.000,A 180.000,B 0.000,C 180.000} C_DIS
LIN {X 97.075,Y 85.983,Z 75.000,A 180.000,B 0.000,C 180.000} C_DIS
LIN {X 96.897,Y 85.989,Z 75.000,A 180.000,B 0.000,C 180.000} C_DIS
LIN {X 96.852,Y 85.992,Z 75.000,A 180.000,B 0.000,C 180.000} C_DIS
LIN {X 96.718,Y 86.001,Z 75.000,A 180.000,B 0.000,C 180.000} C_DIS
LIN {X 96.360,Y 86.031,Z 75.000,A 180.000,B 0.000,C 180.000} C_DIS
LIN {X 96.181,Y 86.047,Z 75.000,A 180.000,B 0.000,C 180.000} C_DIS
LIN {X 96.003,Y 86.072,Z 75.000,A 180.000,B 0.000,C 180.000} C_DIS
LIN {X 95.824,Y 86.097,Z 75.000,A 180.000,B 0.000,C 180.000} C_DIS
LIN {X 95.645,Y 86.123,Z 75.000,A 180.000,B 0.000,C 180.000} C_DIS
LIN {X 95.466,Y 86.155,Z 75.000,A 180.000,B 0.000,C 180.000} C_DIS
LIN {X 95.389,Y 86.170,Z 75.000,A 180.000,B 0.000,C 180.000} C_DIS
LIN {X 95.109,Y 86.226,Z 75.000,A 180.000,B 0.000,C 180.000} C_DIS
LIN {X 94.930,Y 86.262,Z 75.000,A 180.000,B 0.000,C 180.000} C_DIS
LIN {X 94.751,Y 86.307,Z 75.000,A 180.000,B 0.000,C 180.000} C_DIS
LIN {X 94.573,Y 86.353,Z 75.000,A 180.000,B 0.000,C 180.000} C_DIS
LIN {X 94.394,Y 86.399,Z 75.000,A 180.000,B 0.000,C 180.000} C_DIS
LIN {X 94.215,Y 86.452,Z 75.000,A 180.000,B 0.000,C 180.000} C_DIS
LIN {X 93.857,Y 86.566,Z 75.000,A 180.000,B 0.000,C 180.000} C_DIS
LIN {X 93.679,Y 86.624,Z 75.000,A 180.000,B 0.000,C 180.000} C_DIS
LIN {X 93.500,Y 86.691,Z 75.000,A 180.000,B 0.000,C 180.000} C_DIS
LIN {X 93.321,Y 86.759,Z 75.000,A 180.000,B 0.000,C 180.000} C_DIS
LIN {X 93.142,Y 86.827,Z 75.000,A 180.000,B 0.000,C 180.000} C_DIS
LIN {X 93.006,Y 86.885,Z 75.000,A 180.000,B 0.000,C 180.000} C_DIS
LIN {X 92.785,Y 86.984,Z 75.000,A 180.000,B 0.000,C 180.000} C_DIS
LIN {X 92.606,Y 87.065,Z 75.000,A 180.000,B 0.000,C 180.000} C_DIS
LIN {X 92.427,Y 87.149,Z 75.000,A 180.000,B 0.000,C 180.000} C_DIS
LIN {X 92.249,Y 87.241,Z 75.000,A 180.000,B 0.000,C 180.000} C_DIS
LIN {X 92.070,Y 87.333,Z 75.000,A 180.000,B 0.000,C 180.000} C_DIS
LIN {X 91.903,Y 87.422,Z 75.000,A 180.000,B 0.000,C 180.000} C_DIS
LIN {X 91.891,Y 87.429,Z 75.000,A 180.000,B 0.000,C 180.000} C_DIS
LIN {X 91.712,Y 87.534,Z 75.000,A 180.000,B 0.000,C 180.000} C_DIS
LIN {X 91.533,Y 87.639,Z 75.000,A 180.000,B 0.000,C 180.000} C_DIS
LIN {X 91.355,Y 87.748,Z 75.000,A 180.000,B 0.000,C 180.000} C_DIS
LIN {X 91.306,Y 87.779,Z 75.000,A 180.000,B 0.000,C 180.000} C_DIS
LIN {X 91.176,Y 87.865,Z 75.000,A 180.000,B 0.000,C 180.000} C_DIS
LIN {X 90.997,Y 87.985,Z 75.000,A 180.000,B 0.000,C 180.000} C_DIS
LIN {X 90.818,Y 88.106,Z 75.000,A 180.000,B 0.000,C 180.000} C_DIS
LIN {X 90.775,Y 88.137,Z 75.000,A 180.000,B 0.000,C 180.000} C_DIS
LIN {X 90.640,Y 88.239,Z 75.000,A 180.000,B 0.000,C 180.000} C_DIS
LIN {X 90.461,Y 88.373,Z 75.000,A 180.000,B 0.000,C 180.000} C_DIS
LIN {X 90.305,Y 88.494,Z 75.000,A 180.000,B 0.000,C 180.000} C_DIS
LIN {X 90.282,Y 88.513,Z 75.000,A 180.000,B 0.000,C 180.000} C_DIS
LIN {X 90.103,Y 88.663,Z 75.000,A 180.000,B 0.000,C 180.000} C_DIS
LIN {X 89.880,Y 88.852,Z 75.000,A 180.000,B 0.000,C 180.000} C_DIS
LIN {X 89.746,Y 88.971,Z 75.000,A 180.000,B 0.000,C 180.000} C_DIS
LIN {X 89.493,Y 89.209,Z 75.000,A 180.000,B 0.000,C 180.000} C_DIS
LIN {X 89.388,Y 89.309,Z 75.000,A 180.000,B 0.000,C 180.000} C_DIS
LIN {X 89.311,Y 89.388,Z 75.000,A 180.000,B 0.000,C 180.000} C_DIS
LIN {X 89.031,Y 89.684,Z 75.000,A 180.000,B 0.000,C 180.000} C_DIS
LIN {X 88.973,Y 89.746,Z 75.000,A 180.000,B 0.000,C 180.000} C_DIS
LIN {X 88.852,Y 89.878,Z 75.000,A 180.000,B 0.000,C 180.000} C_DIS
LIN {X 88.813,Y 89.925,Z 75.000,A 180.000,B 0.000,C 180.000} C_DIS
LIN {X 88.662,Y 90.103,Z 75.000,A 180.000,B 0.000,C 180.000} C_DIS
LIN {X 88.511,Y 90.282,Z 75.000,A 180.000,B 0.000,C 180.000} C_DIS
LIN {X 88.494,Y 90.303,Z 75.000,A 180.000,B 0.000,C 180.000} C_DIS
LIN {X 88.374,Y 90.461,Z 75.000,A 180.000,B 0.000,C 180.000} C_DIS
LIN {X 88.240,Y 90.640,Z 75.000,A 180.000,B 0.000,C 180.000} C_DIS
LIN {X 88.137,Y 90.778,Z 75.000,A 180.000,B 0.000,C 180.000} C_DIS
LIN {X 88.107,Y 90.818,Z 75.000,A 180.000,B 0.000,C 180.000} C_DIS
LIN {X 87.984,Y 90.997,Z 75.000,A 180.000,B 0.000,C 180.000} C_DIS
LIN {X 87.832,Y 91.225,Z 75.000,A 180.000,B 0.000,C 180.000} C_DIS
LIN {X 87.779,Y 91.304,Z 75.000,A 180.000,B 0.000,C 180.000} C_DIS
LIN {X 87.746,Y 91.355,Z 75.000,A 180.000,B 0.000,C 180.000} C_DIS
LIN {X 87.639,Y 91.533,Z 75.000,A 180.000,B 0.000,C 180.000} C_DIS
LIN {X 87.534,Y 91.712,Z 75.000,A 180.000,B 0.000,C 180.000} C_DIS
LIN {X 87.430,Y 91.891,Z 75.000,A 180.000,B 0.000,C 180.000} C_DIS
LIN {X 87.422,Y 91.906,Z 75.000,A 180.000,B 0.000,C 180.000} C_DIS
LIN {X 87.334,Y 92.070,Z 75.000,A 180.000,B 0.000,C 180.000} C_DIS
LIN {X 87.149,Y 92.427,Z 75.000,A 180.000,B 0.000,C 180.000} C_DIS
LIN {X 87.064,Y 92.605,Z 75.000,A 180.000,B 0.000,C 180.000} C_DIS
LIN {X 86.904,Y 92.964,Z 75.000,A 180.000,B 0.000,C 180.000} C_DIS
LIN {X 86.885,Y 93.005,Z 75.000,A 180.000,B 0.000,C 180.000} C_DIS
LIN {X 86.829,Y 93.142,Z 75.000,A 180.000,B 0.000,C 180.000} C_DIS
LIN {X 86.760,Y 93.321,Z 75.000,A 180.000,B 0.000,C 180.000} C_DIS
LIN {X 86.692,Y 93.500,Z 75.000,A 180.000,B 0.000,C 180.000} C_DIS
LIN {X 86.624,Y 93.679,Z 75.000,A 180.000,B 0.000,C 180.000} C_DIS
LIN {X 86.565,Y 93.857,Z 75.000,A 180.000,B 0.000,C 180.000} C_DIS
LIN {X 86.451,Y 94.215,Z 75.000,A 180.000,B 0.000,C 180.000} C_DIS
LIN {X 86.401,Y 94.394,Z 75.000,A 180.000,B 0.000,C 180.000} C_DIS
LIN {X 86.308,Y 94.751,Z 75.000,A 180.000,B 0.000,C 180.000} C_DIS
LIN {X 86.263,Y 94.930,Z 75.000,A 180.000,B 0.000,C 180.000} C_DIS
LIN {X 86.225,Y 95.109,Z 75.000,A 180.000,B 0.000,C 180.000} C_DIS
LIN {X 86.154,Y 95.466,Z 75.000,A 180.000,B 0.000,C 180.000} C_DIS
LIN {X 86.123,Y 95.645,Z 75.000,A 180.000,B 0.000,C 180.000} C_DIS
LIN {X 86.073,Y 96.003,Z 75.000,A 180.000,B 0.000,C 180.000} C_DIS
LIN {X 86.052,Y 96.163,Z 75.000,A 180.000,B 0.000,C 180.000} C_DIS
LIN {X 86.049,Y 96.181,Z 75.000,A 180.000,B 0.000,C 180.000} C_DIS
LIN {X 86.030,Y 96.360,Z 75.000,A 180.000,B 0.000,C 180.000} C_DIS
LIN {X 86.000,Y 96.718,Z 75.000,A 180.000,B 0.000,C 180.000} C_DIS
LIN {X 85.992,Y 96.825,Z 75.000,A 180.000,B 0.000,C 180.000} C_DIS
LIN {X 85.988,Y 96.897,Z 75.000,A 180.000,B 0.000,C 180.000} C_DIS
LIN {X 85.983,Y 97.075,Z 75.000,A 180.000,B 0.000,C 180.000} C_DIS
LIN {X 85.978,Y 97.254,Z 75.000,A 180.000,B 0.000,C 180.000} C_DIS
LIN {X 85.973,Y 97.433,Z 75.000,A 180.000,B 0.000,C 180.000} C_DIS
LIN {X 85.974,Y 97.612,Z 75.000,A 180.000,B 0.000,C 180.000} C_DIS
LIN {X 85.979,Y 97.790,Z 75.000,A 180.000,B 0.000,C 180.000} C_DIS
LIN {X 85.984,Y 97.969,Z 75.000,A 180.000,B 0.000,C 180.000} C_DIS
LIN {X 85.990,Y 98.148,Z 75.000,A 180.000,B 0.000,C 180.000} C_DIS
LIN {X 85.992,Y 98.175,Z 75.000,A 180.000,B 0.000,C 180.000} C_DIS
LIN {X 86.004,Y 98.327,Z 75.000,A 180.000,B 0.000,C 180.000} C_DIS
LIN {X 86.034,Y 98.684,Z 75.000,A 180.000,B 0.000,C 180.000} C_DIS
LIN {X 86.055,Y 98.863,Z 75.000,A 180.000,B 0.000,C 180.000} C_DIS
LIN {X 86.079,Y 99.042,Z 75.000,A 180.000,B 0.000,C 180.000} C_DIS
LIN {X 86.105,Y 99.221,Z 75.000,A 180.000,B 0.000,C 180.000} C_DIS
LIN {X 86.130,Y 99.399,Z 75.000,A 180.000,B 0.000,C 180.000} C_DIS
LIN {X 86.162,Y 99.578,Z 75.000,A 180.000,B 0.000,C 180.000} C_DIS
LIN {X 86.234,Y 99.936,Z 75.000,A 180.000,B 0.000,C 180.000} C_DIS
LIN {X 86.274,Y 100.114,Z 75.000,A 180.000,B 0.000,C 180.000} C_DIS
LIN {X 86.320,Y 100.293,Z 75.000,A 180.000,B 0.000,C 180.000} C_DIS
LIN {X 86.412,Y 100.651,Z 75.000,A 180.000,B 0.000,C 180.000} C_DIS
LIN {X 86.465,Y 100.829,Z 75.000,A 180.000,B 0.000,C 180.000} C_DIS
LIN {X 86.579,Y 101.187,Z 75.000,A 180.000,B 0.000,C 180.000} C_DIS
LIN {X 86.641,Y 101.366,Z 75.000,A 180.000,B 0.000,C 180.000} C_DIS
LIN {X 86.777,Y 101.723,Z 75.000,A 180.000,B 0.000,C 180.000} C_DIS
LIN {X 86.847,Y 101.902,Z 75.000,A 180.000,B 0.000,C 180.000} C_DIS
LIN {X 86.885,Y 101.995,Z 75.000,A 180.000,B 0.000,C 180.000} C_DIS
LIN {X 86.924,Y 102.081,Z 75.000,A 180.000,B 0.000,C 180.000} C_DIS
LIN {X 87.064,Y 102.395,Z 75.000,A 180.000,B 0.000,C 180.000} C_DIS
LIN {X 87.084,Y 102.438,Z 75.000,A 180.000,B 0.000,C 180.000} C_DIS
LIN {X 87.172,Y 102.617,Z 75.000,A 180.000,B 0.000,C 180.000} C_DIS
LIN {X 87.264,Y 102.796,Z 75.000,A 180.000,B 0.000,C 180.000} C_DIS
LIN {X 87.357,Y 102.975,Z 75.000,A 180.000,B 0.000,C 180.000} C_DIS
LIN {X 87.422,Y 103.094,Z 75.000,A 180.000,B 0.000,C 180.000} C_DIS
LIN {X 87.455,Y 103.153,Z 75.000,A 180.000,B 0.000,C 180.000} C_DIS
LIN {X 87.560,Y 103.332,Z 75.000,A 180.000,B 0.000,C 180.000} C_DIS
LIN {X 87.665,Y 103.511,Z 75.000,A 180.000,B 0.000,C 180.000} C_DIS
LIN {X 87.775,Y 103.690,Z 75.000,A 180.000,B 0.000,C 180.000} C_DIS
LIN {X 87.779,Y 103.696,Z 75.000,A 180.000,B 0.000,C 180.000} C_DIS
LIN {X 88.014,Y 104.047,Z 75.000,A 180.000,B 0.000,C 180.000} C_DIS
LIN {X 88.137,Y 104.222,Z 75.000,A 180.000,B 0.000,C 180.000} C_DIS
LIN {X 88.140,Y 104.226,Z 75.000,A 180.000,B 0.000,C 180.000} C_DIS
LIN {X 88.273,Y 104.405,Z 75.000,A 180.000,B 0.000,C 180.000} C_DIS
LIN {X 88.408,Y 104.584,Z 75.000,A 180.000,B 0.000,C 180.000} C_DIS
LIN {X 88.494,Y 104.697,Z 75.000,A 180.000,B 0.000,C 180.000} C_DIS
LIN {X 88.548,Y 104.762,Z 75.000,A 180.000,B 0.000,C 180.000} C_DIS
LIN {X 88.699,Y 104.941,Z 75.000,A 180.000,B 0.000,C 180.000} C_DIS
LIN {X 88.850,Y 105.120,Z 75.000,A 180.000,B 0.000,C 180.000} C_DIS
LIN {X 88.852,Y 105.122,Z 75.000,A 180.000,B 0.000,C 180.000} C_DIS
LIN {X 89.015,Y 105.299,Z 75.000,A 180.000,B 0.000,C 180.000} C_DIS
LIN {X 89.209,Y 105.505,Z 75.000,A 180.000,B 0.000,C 180.000} C_DIS
LIN {X 89.354,Y 105.656,Z 75.000,A 180.000,B 0.000,C 180.000} C_DIS
LIN {X 89.388,Y 105.691,Z 75.000,A 180.000,B 0.000,C 180.000} C_DIS
LIN {X 89.540,Y 105.835,Z 75.000,A 180.000,B 0.000,C 180.000} C_DIS
LIN {X 89.746,Y 106.029,Z 75.000,A 180.000,B 0.000,C 180.000} C_DIS
LIN {X 89.925,Y 106.186,Z 75.000,A 180.000,B 0.000,C 180.000} C_DIS
LIN {X 90.144,Y 106.371,Z 75.000,A 180.000,B 0.000,C 180.000} C_DIS
LIN {X 90.282,Y 106.487,Z 75.000,A 180.000,B 0.000,C 180.000} C_DIS
LIN {X 90.360,Y 106.550,Z 75.000,A 180.000,B 0.000,C 180.000} C_DIS
LIN {X 90.461,Y 106.627,Z 75.000,A 180.000,B 0.000,C 180.000} C_DIS
LIN {X 90.640,Y 106.761,Z 75.000,A 180.000,B 0.000,C 180.000} C_DIS
LIN {X 90.818,Y 106.894,Z 75.000,A 180.000,B 0.000,C 180.000} C_DIS
LIN {X 90.837,Y 106.908,Z 75.000,A 180.000,B 0.000,C 180.000} C_DIS
LIN {X 90.997,Y 107.015,Z 75.000,A 180.000,B 0.000,C 180.000} C_DIS
LIN {X 91.176,Y 107.135,Z 75.000,A 180.000,B 0.000,C 180.000} C_DIS
LIN {X 91.355,Y 107.252,Z 75.000,A 180.000,B 0.000,C 180.000} C_DIS
LIN {X 91.376,Y 107.265,Z 75.000,A 180.000,B 0.000,C 180.000} C_DIS
LIN {X 91.533,Y 107.361,Z 75.000,A 180.000,B 0.000,C 180.000} C_DIS
LIN {X 91.712,Y 107.466,Z 75.000,A 180.000,B 0.000,C 180.000} C_DIS
LIN {X 91.891,Y 107.571,Z 75.000,A 180.000,B 0.000,C 180.000} C_DIS
LIN {X 91.985,Y 107.623,Z 75.000,A 180.000,B 0.000,C 180.000} C_DIS
LIN {X 92.331,Y 107.802,Z 75.000,A 180.000,B 0.000,C 180.000} C_DIS
LIN {X 92.427,Y 107.851,Z 75.000,A 180.000,B 0.000,C 180.000} C_DIS
LIN {X 92.606,Y 107.935,Z 75.000,A 180.000,B 0.000,C 180.000} C_DIS
LIN {X 92.706,Y 107.980,Z 75.000,A 180.000,B 0.000,C 180.000} C_DIS
LIN {X 92.964,Y 108.096,Z 75.000,A 180.000,B 0.000,C 180.000} C_DIS
LIN {X 93.109,Y 108.159,Z 75.000,A 180.000,B 0.000,C 180.000} C_DIS
LIN {X 93.142,Y 108.173,Z 75.000,A 180.000,B 0.000,C 180.000} C_DIS
LIN {X 93.321,Y 108.241,Z 75.000,A 180.000,B 0.000,C 180.000} C_DIS
LIN {X 93.575,Y 108.338,Z 75.000,A 180.000,B 0.000,C 180.000} C_DIS
LIN {X 93.679,Y 108.376,Z 75.000,A 180.000,B 0.000,C 180.000} C_DIS
LIN {X 93.857,Y 108.434,Z 75.000,A 180.000,B 0.000,C 180.000} C_DIS
LIN {X 94.215,Y 108.548,Z 75.000,A 180.000,B 0.000,C 180.000} C_DIS
LIN {X 94.394,Y 108.601,Z 75.000,A 180.000,B 0.000,C 180.000} C_DIS
LIN {X 94.573,Y 108.647,Z 75.000,A 180.000,B 0.000,C 180.000} C_DIS
LIN {X 94.759,Y 108.695,Z 75.000,A 180.000,B 0.000,C 180.000} C_DIS
LIN {X 94.930,Y 108.738,Z 75.000,A 180.000,B 0.000,C 180.000} C_DIS
LIN {X 95.109,Y 108.774,Z 75.000,A 180.000,B 0.000,C 180.000} C_DIS
LIN {X 95.288,Y 108.809,Z 75.000,A 180.000,B 0.000,C 180.000} C_DIS
LIN {X 95.466,Y 108.845,Z 75.000,A 180.000,B 0.000,C 180.000} C_DIS
LIN {X 95.625,Y 108.874,Z 75.000,A 180.000,B 0.000,C 180.000} C_DIS
LIN {X 95.645,Y 108.877,Z 75.000,A 180.000,B 0.000,C 180.000} C_DIS
LIN {X 95.824,Y 108.903,Z 75.000,A 180.000,B 0.000,C 180.000} C_DIS
LIN {X 96.003,Y 108.928,Z 75.000,A 180.000,B 0.000,C 180.000} C_DIS
LIN {X 96.181,Y 108.953,Z 75.000,A 180.000,B 0.000,C 180.000} C_DIS
LIN {X 96.360,Y 108.969,Z 75.000,A 180.000,B 0.000,C 180.000} C_DIS
LIN {X 96.718,Y 108.999,Z 75.000,A 180.000,B 0.000,C 180.000} C_DIS
LIN {X 96.897,Y 109.011,Z 75.000,A 180.000,B 0.000,C 180.000} C_DIS
LIN {X 97.075,Y 109.017,Z 75.000,A 180.000,B 0.000,C 180.000} C_DIS
LIN {X 97.433,Y 109.027,Z 75.000,A 180.000,B 0.000,C 180.000} C_DIS
LIN {X 97.612,Y 109.026,Z 75.000,A 180.000,B 0.000,C 180.000} C_DIS
LIN {X 97.969,Y 109.016,Z 75.000,A 180.000,B 0.000,C 180.000} C_DIS
LIN {X 98.148,Y 109.008,Z 75.000,A 180.000,B 0.000,C 180.000} C_DIS
LIN {X 98.327,Y 108.996,Z 75.000,A 180.000,B 0.000,C 180.000} C_DIS
LIN {X 98.684,Y 108.965,Z 75.000,A 180.000,B 0.000,C 180.000} C_DIS
LIN {X 98.863,Y 108.947,Z 75.000,A 180.000,B 0.000,C 180.000} C_DIS
LIN {X 99.042,Y 108.922,Z 75.000,A 180.000,B 0.000,C 180.000} C_DIS
LIN {X 99.221,Y 108.896,Z 75.000,A 180.000,B 0.000,C 180.000} C_DIS
LIN {X 99.375,Y 108.874,Z 75.000,A 180.000,B 0.000,C 180.000} C_DIS
LIN {X 99.399,Y 108.870,Z 75.000,A 180.000,B 0.000,C 180.000} C_DIS
LIN {X 99.578,Y 108.836,Z 75.000,A 180.000,B 0.000,C 180.000} C_DIS
LIN {X 99.936,Y 108.765,Z 75.000,A 180.000,B 0.000,C 180.000} C_DIS
LIN {X 100.114,Y 108.728,Z 75.000,A 180.000,B 0.000,C 180.000} C_DIS
LIN {X 100.241,Y 108.695,Z 75.000,A 180.000,B 0.000,C 180.000} C_DIS
LIN {X 100.472,Y 108.636,Z 75.000,A 180.000,B 0.000,C 180.000} C_DIS
LIN {X 100.651,Y 108.589,Z 75.000,A 180.000,B 0.000,C 180.000} C_DIS
LIN {X 100.829,Y 108.534,Z 75.000,A 180.000,B 0.000,C 180.000} C_DIS
LIN {X 101.008,Y 108.477,Z 75.000,A 180.000,B 0.000,C 180.000} C_DIS
LIN {X 101.187,Y 108.420,Z 75.000,A 180.000,B 0.000,C 180.000} C_DIS
LIN {X 101.366,Y 108.360,Z 75.000,A 180.000,B 0.000,C 180.000} C_DIS
LIN {X 101.425,Y 108.338,Z 75.000,A 180.000,B 0.000,C 180.000} C_DIS
LIN {X 101.723,Y 108.224,Z 75.000,A 180.000,B 0.000,C 180.000} C_DIS
LIN {X 101.891,Y 108.159,Z 75.000,A 180.000,B 0.000,C 180.000} C_DIS
LIN {X 101.902,Y 108.155,Z 75.000,A 180.000,B 0.000,C 180.000} C_DIS
LIN {X 102.081,Y 108.076,Z 75.000,A 180.000,B 0.000,C 180.000} C_DIS
LIN {X 102.294,Y 107.980,Z 75.000,A 180.000,B 0.000,C 180.000} C_DIS
LIN {X 102.438,Y 107.915,Z 75.000,A 180.000,B 0.000,C 180.000} C_DIS
LIN {X 102.617,Y 107.828,Z 75.000,A 180.000,B 0.000,C 180.000} C_DIS
LIN {X 103.015,Y 107.623,Z 75.000,A 180.000,B 0.000,C 180.000} C_DIS
LIN {X 103.153,Y 107.545,Z 75.000,A 180.000,B 0.000,C 180.000} C_DIS
LIN {X 103.511,Y 107.335,Z 75.000,A 180.000,B 0.000,C 180.000} C_DIS
LIN {X 103.624,Y 107.265,Z 75.000,A 180.000,B 0.000,C 180.000} C_DIS
LIN {X 103.690,Y 107.224,Z 75.000,A 180.000,B 0.000,C 180.000} C_DIS
LIN {X 103.869,Y 107.105,Z 75.000,A 180.000,B 0.000,C 180.000} C_DIS
LIN {X 104.047,Y 106.986,Z 75.000,A 180.000,B 0.000,C 180.000} C_DIS
LIN {X 104.163,Y 106.908,Z 75.000,A 180.000,B 0.000,C 180.000} C_DIS
LIN {X 104.226,Y 106.862,Z 75.000,A 180.000,B 0.000,C 180.000} C_DIS
LIN {X 104.405,Y 106.728,Z 75.000,A 180.000,B 0.000,C 180.000} C_DIS
LIN {X 104.584,Y 106.593,Z 75.000,A 180.000,B 0.000,C 180.000} C_DIS
LIN {X 104.640,Y 106.550,Z 75.000,A 180.000,B 0.000,C 180.000} C_DIS
LIN {X 104.762,Y 106.450,Z 75.000,A 180.000,B 0.000,C 180.000} C_DIS
LIN {X 104.856,Y 106.371,Z 75.000,A 180.000,B 0.000,C 180.000} C_DIS
LIN {X 105.120,Y 106.148,Z 75.000,A 180.000,B 0.000,C 180.000} C_DIS
LIN {X 105.271,Y 106.014,Z 75.000,A 180.000,B 0.000,C 180.000} C_DIS
LIN {X 105.477,Y 105.818,Z 75.000,A 180.000,B 0.000,C 180.000} C_DIS
LIN {X 105.646,Y 105.656,Z 75.000,A 180.000,B 0.000,C 180.000} C_DIS
LIN {X 105.656,Y 105.646,Z 75.000,A 180.000,B 0.000,C 180.000} C_DIS
LIN {X 105.816,Y 105.477,Z 75.000,A 180.000,B 0.000,C 180.000} C_DIS
LIN {X 105.985,Y 105.299,Z 75.000,A 180.000,B 0.000,C 180.000} C_DIS
LIN {X 106.014,Y 105.268,Z 75.000,A 180.000,B 0.000,C 180.000} C_DIS
LIN {X 106.150,Y 105.120,Z 75.000,A 180.000,B 0.000,C 180.000} C_DIS
LIN {X 106.193,Y 105.069,Z 75.000,A 180.000,B 0.000,C 180.000} C_DIS
LIN {X 106.452,Y 104.762,Z 75.000,A 180.000,B 0.000,C 180.000} C_DIS
LIN {X 106.550,Y 104.639,Z 75.000,A 180.000,B 0.000,C 180.000} C_DIS
LIN {X 106.729,Y 104.402,Z 75.000,A 180.000,B 0.000,C 180.000} C_DIS
LIN {X 106.860,Y 104.226,Z 75.000,A 180.000,B 0.000,C 180.000} C_DIS
LIN {X 106.908,Y 104.161,Z 75.000,A 180.000,B 0.000,C 180.000} C_DIS
LIN {X 106.986,Y 104.047,Z 75.000,A 180.000,B 0.000,C 180.000} C_DIS
LIN {X 107.225,Y 103.690,Z 75.000,A 180.000,B 0.000,C 180.000} C_DIS
LIN {X 107.265,Y 103.627,Z 75.000,A 180.000,B 0.000,C 180.000} C_DIS
LIN {X 107.335,Y 103.511,Z 75.000,A 180.000,B 0.000,C 180.000} C_DIS
LIN {X 107.444,Y 103.325,Z 75.000,A 180.000,B 0.000,C 180.000} C_DIS
LIN {X 107.545,Y 103.153,Z 75.000,A 180.000,B 0.000,C 180.000} C_DIS
LIN {X 107.623,Y 103.013,Z 75.000,A 180.000,B 0.000,C 180.000} C_DIS
LIN {X 107.643,Y 102.975,Z 75.000,A 180.000,B 0.000,C 180.000} C_DIS
LIN {X 107.736,Y 102.796,Z 75.000,A 180.000,B 0.000,C 180.000} C_DIS
LIN {X 107.828,Y 102.617,Z 75.000,A 180.000,B 0.000,C 180.000} C_DIS
LIN {X 107.916,Y 102.438,Z 75.000,A 180.000,B 0.000,C 180.000} C_DIS
LIN {X 107.965,Y 102.330,Z 75.000,A 180.000,B 0.000,C 180.000} C_DIS
; Link Move Starts
LIN {X 108.094,Y 102.043,Z 75.000,A 180.000,B 0.000,C 180.000} C_DIS
LIN {X 108.209,Y 101.763,Z 74.998,A 180.000,B 0.000,C 180.000} C_DIS
LIN {X 108.322,Y 101.469,Z 74.996,A 180.000,B 0.000,C 180.000} C_DIS
LIN {X 108.426,Y 101.184,Z 74.993,A 180.000,B 0.000,C 180.000} C_DIS
LIN {X 108.523,Y 100.886,Z 74.989,A 180.000,B 0.000,C 180.000} C_DIS
LIN {X 108.610,Y 100.593,Z 74.984,A 180.000,B 0.000,C 180.000} C_DIS
LIN {X 108.651,Y 100.443,Z 74.981,A 180.000,B 0.000,C 180.000} C_DIS
LIN {X 108.691,Y 100.292,Z 74.978,A 180.000,B 0.000,C 180.000} C_DIS
LIN {X 108.730,Y 100.144,Z 74.975,A 180.000,B 0.000,C 180.000} C_DIS
LIN {X 108.767,Y 99.997,Z 74.972,A 180.000,B 0.000,C 180.000} C_DIS
LIN {X 108.799,Y 99.844,Z 74.969,A 180.000,B 0.000,C 180.000} C_DIS
LIN {X 108.832,Y 99.690,Z 74.965,A 180.000,B 0.000,C 180.000} C_DIS
LIN {X 108.863,Y 99.539,Z 74.962,A 180.000,B 0.000,C 180.000} C_DIS
LIN {X 108.892,Y 99.387,Z 74.958,A 180.000,B 0.000,C 180.000} C_DIS
LIN {X 108.915,Y 99.234,Z 74.954,A 180.000,B 0.000,C 180.000} C_DIS
LIN {X 108.939,Y 99.082,Z 74.950,A 180.000,B 0.000,C 180.000} C_DIS
LIN {X 108.962,Y 98.929,Z 74.945,A 180.000,B 0.000,C 180.000} C_DIS
LIN {X 108.984,Y 98.777,Z 74.941,A 180.000,B 0.000,C 180.000} C_DIS
LIN {X 109.001,Y 98.622,Z 74.936,A 180.000,B 0.000,C 180.000} C_DIS
LIN {X 109.016,Y 98.468,Z 74.932,A 180.000,B 0.000,C 180.000} C_DIS
LIN {X 109.032,Y 98.313,Z 74.927,A 180.000,B 0.000,C 180.000} C_DIS
LIN {X 109.039,Y 98.235,Z 74.924,A 180.000,B 0.000,C 180.000} C_DIS
LIN {X 109.046,Y 98.157,Z 74.922,A 180.000,B 0.000,C 180.000} C_DIS
LIN {X 109.051,Y 98.080,Z 74.919,A 180.000,B 0.000,C 180.000} C_DIS
LIN {X 109.054,Y 98.004,Z 74.917,A 180.000,B 0.000,C 180.000} C_DIS
LIN {X 109.057,Y 97.927,Z 74.914,A 180.000,B 0.000,C 180.000} C_DIS
LIN {X 109.061,Y 97.851,Z 74.911,A 180.000,B 0.000,C 180.000} C_DIS
LIN {X 109.064,Y 97.773,Z 74.909,A 180.000,B 0.000,C 180.000} C_DIS
LIN {X 109.067,Y 97.696,Z 74.906,A 180.000,B 0.000,C 180.000} C_DIS
LIN {X 109.071,Y 97.618,Z 74.903,A 180.000,B 0.000,C 180.000} C_DIS
LIN {X 109.073,Y 97.540,Z 74.901,A 180.000,B 0.000,C 180.000} C_DIS
LIN {X 109.074,Y 97.463,Z 74.898,A 180.000,B 0.000,C 180.000} C_DIS
LIN {X 109.075,Y 97.386,Z 74.895,A 180.000,B 0.000,C 180.000} C_DIS
LIN {X 109.074,Y 97.309,Z 74.893,A 180.000,B 0.000,C 180.000} C_DIS
LIN {X 109.073,Y 97.231,Z 74.890,A 180.000,B 0.000,C 180.000} C_DIS
LIN {X 109.072,Y 97.153,Z 74.887,A 180.000,B 0.000,C 180.000} C_DIS
LIN {X 109.071,Y 97.074,Z 74.884,A 180.000,B 0.000,C 180.000} C_DIS
LIN {X 109.070,Y 96.995,Z 74.882,A 180.000,B 0.000,C 180.000} C_DIS
LIN {X 109.069,Y 96.916,Z 74.879,A 180.000,B 0.000,C 180.000} C_DIS
LIN {X 109.067,Y 96.840,Z 74.876,A 180.000,B 0.000,C 180.000} C_DIS
LIN {X 109.063,Y 96.764,Z 74.874,A 180.000,B 0.000,C 180.000} C_DIS
LIN {X 109.058,Y 96.688,Z 74.871,A 180.000,B 0.000,C 180.000} C_DIS
LIN {X 109.053,Y 96.611,Z 74.868,A 180.000,B 0.000,C 180.000} C_DIS
LIN {X 109.047,Y 96.533,Z 74.865,A 180.000,B 0.000,C 180.000} C_DIS
LIN {X 109.042,Y 96.455,Z 74.863,A 180.000,B 0.000,C 180.000} C_DIS
LIN {X 109.037,Y 96.377,Z 74.860,A 180.000,B 0.000,C 180.000} C_DIS
LIN {X 109.031,Y 96.299,Z 74.857,A 180.000,B 0.000,C 180.000} C_DIS
LIN {X 109.024,Y 96.223,Z 74.855,A 180.000,B 0.000,C 180.000} C_DIS
LIN {X 109.016,Y 96.146,Z 74.852,A 180.000,B 0.000,C 180.000} C_DIS
LIN {X 109.007,Y 96.069,Z 74.849,A 180.000,B 0.000,C 180.000} C_DIS
LIN {X 108.998,Y 95.993,Z 74.846,A 180.000,B 0.000,C 180.000} C_DIS
LIN {X 108.978,Y 95.837,Z 74.841,A 180.000,B 0.000,C 180.000} C_DIS
LIN {X 108.949,Y 95.604,Z 74.833,A 180.000,B 0.000,C 180.000} C_DIS
LIN {X 108.939,Y 95.528,Z 74.830,A 180.000,B 0.000,C 180.000} C_DIS
LIN {X 108.926,Y 95.453,Z 74.827,A 180.000,B 0.000,C 180.000} C_DIS
LIN {X 108.912,Y 95.377,Z 74.825,A 180.000,B 0.000,C 180.000} C_DIS
LIN {X 108.884,Y 95.223,Z 74.819,A 180.000,B 0.000,C 180.000} C_DIS
LIN {X 108.856,Y 95.068,Z 74.814,A 180.000,B 0.000,C 180.000} C_DIS
LIN {X 108.842,Y 94.992,Z 74.811,A 180.000,B 0.000,C 180.000} C_DIS
LIN {X 108.826,Y 94.917,Z 74.808,A 180.000,B 0.000,C 180.000} C_DIS
LIN {X 108.809,Y 94.842,Z 74.806,A 180.000,B 0.000,C 180.000} C_DIS
LIN {X 108.791,Y 94.768,Z 74.803,A 180.000,B 0.000,C 180.000} C_DIS
LIN {X 108.754,Y 94.614,Z 74.798,A 180.000,B 0.000,C 180.000} C_DIS
LIN {X 108.699,Y 94.386,Z 74.789,A 180.000,B 0.000,C 180.000} C_DIS
LIN {X 108.681,Y 94.311,Z 74.787,A 180.000,B 0.000,C 180.000} C_DIS
LIN {X 108.661,Y 94.237,Z 74.784,A 180.000,B 0.000,C 180.000} C_DIS
LIN {X 108.640,Y 94.163,Z 74.781,A 180.000,B 0.000,C 180.000} C_DIS
LIN {X 108.572,Y 93.937,Z 74.773,A 180.000,B 0.000,C 180.000} C_DIS
LIN {X 108.527,Y 93.788,Z 74.768,A 180.000,B 0.000,C 180.000} C_DIS
LIN {X 108.504,Y 93.713,Z 74.765,A 180.000,B 0.000,C 180.000} C_DIS
LIN {X 108.480,Y 93.640,Z 74.762,A 180.000,B 0.000,C 180.000} C_DIS
LIN {X 108.454,Y 93.567,Z 74.759,A 180.000,B 0.000,C 180.000} C_DIS
LIN {X 108.320,Y 93.199,Z 74.746,A 180.000,B 0.000,C 180.000} C_DIS
LIN {X 108.293,Y 93.127,Z 74.743,A 180.000,B 0.000,C 180.000} C_DIS
LIN {X 108.266,Y 93.054,Z 74.740,A 180.000,B 0.000,C 180.000} C_DIS
LIN {X 108.238,Y 92.982,Z 74.738,A 180.000,B 0.000,C 180.000} C_DIS
LIN {X 108.208,Y 92.910,Z 74.735,A 180.000,B 0.000,C 180.000} C_DIS
LIN {X 108.054,Y 92.551,Z 74.721,A 180.000,B 0.000,C 180.000} C_DIS
LIN {X 108.023,Y 92.479,Z 74.719,A 180.000,B 0.000,C 180.000} C_DIS
LIN {X 107.990,Y 92.409,Z 74.716,A 180.000,B 0.000,C 180.000} C_DIS
LIN {X 107.956,Y 92.339,Z 74.713,A 180.000,B 0.000,C 180.000} C_DIS
LIN {X 107.781,Y 91.988,Z 74.699,A 180.000,B 0.000,C 180.000} C_DIS
LIN {X 107.746,Y 91.918,Z 74.697,A 180.000,B 0.000,C 180.000} C_DIS
LIN {X 107.710,Y 91.849,Z 74.694,A 180.000,B 0.000,C 180.000} C_DIS
LIN {X 107.673,Y 91.780,Z 74.691,A 180.000,B 0.000,C 180.000} C_DIS
LIN {X 107.635,Y 91.712,Z 74.689,A 180.000,B 0.000,C 180.000} C_DIS
LIN {X 107.518,Y 91.507,Z 74.680,A 180.000,B 0.000,C 180.000} C_DIS
LIN {X 107.441,Y 91.371,Z 74.675,A 180.000,B 0.000,C 180.000} C_DIS
LIN {X 107.402,Y 91.303,Z 74.672,A 180.000,B 0.000,C 180.000} C_DIS
LIN {X 107.361,Y 91.236,Z 74.669,A 180.000,B 0.000,C 180.000} C_DIS
LIN {X 107.319,Y 91.171,Z 74.667,A 180.000,B 0.000,C 180.000} C_DIS
LIN {X 107.192,Y 90.974,Z 74.659,A 180.000,B 0.000,C 180.000} C_DIS
LIN {X 107.107,Y 90.842,Z 74.653,A 180.000,B 0.000,C 180.000} C_DIS
LIN {X 107.064,Y 90.777,Z 74.650,A 180.000,B 0.000,C 180.000} C_DIS
LIN {X 107.019,Y 90.713,Z 74.648,A 180.000,B 0.000,C 180.000} C_DIS
LIN {X 106.974,Y 90.649,Z 74.645,A 180.000,B 0.000,C 180.000} C_DIS
LIN {X 106.928,Y 90.585,Z 74.642,A 180.000,B 0.000,C 180.000} C_DIS
LIN {X 106.882,Y 90.522,Z 74.639,A 180.000,B 0.000,C 180.000} C_DIS
LIN {X 106.836,Y 90.458,Z 74.637,A 180.000,B 0.000,C 180.000} C_DIS
LIN {X 106.789,Y 90.395,Z 74.634,A 180.000,B 0.000,C 180.000} C_DIS
LIN {X 106.743,Y 90.331,Z 74.631,A 180.000,B 0.000,C 180.000} C_DIS
LIN {X 106.697,Y 90.267,Z 74.628,A 180.000,B 0.000,C 180.000} C_DIS
LIN {X 106.651,Y 90.205,Z 74.626,A 180.000,B 0.000,C 180.000} C_DIS
LIN {X 106.602,Y 90.143,Z 74.623,A 180.000,B 0.000,C 180.000} C_DIS
LIN {X 106.553,Y 90.083,Z 74.620,A 180.000,B 0.000,C 180.000} C_DIS
LIN {X 106.504,Y 90.023,Z 74.618,A 180.000,B 0.000,C 180.000} C_DIS
LIN {X 106.454,Y 89.962,Z 74.615,A 180.000,B 0.000,C 180.000} C_DIS
LIN {X 106.404,Y 89.901,Z 74.612,A 180.000,B 0.000,C 180.000} C_DIS
LIN {X 106.354,Y 89.840,Z 74.609,A 180.000,B 0.000,C 180.000} C_DIS
LIN {X 106.304,Y 89.779,Z 74.607,A 180.000,B 0.000,C 180.000} C_DIS
LIN {X 106.254,Y 89.719,Z 74.604,A 180.000,B 0.000,C 180.000} C_DIS
LIN {X 106.202,Y 89.661,Z 74.601,A 180.000,B 0.000,C 180.000} C_DIS
LIN {X 106.150,Y 89.603,Z 74.598,A 180.000,B 0.000,C 180.000} C_DIS
LIN {X 106.097,Y 89.545,Z 74.596,A 180.000,B 0.000,C 180.000} C_DIS
LIN {X 106.044,Y 89.487,Z 74.593,A 180.000,B 0.000,C 180.000} C_DIS
LIN {X 105.991,Y 89.429,Z 74.590,A 180.000,B 0.000,C 180.000} C_DIS
LIN {X 105.937,Y 89.371,Z 74.587,A 180.000,B 0.000,C 180.000} C_DIS
LIN {X 105.884,Y 89.313,Z 74.585,A 180.000,B 0.000,C 180.000} C_DIS
LIN {X 105.831,Y 89.255,Z 74.582,A 180.000,B 0.000,C 180.000} C_DIS
LIN {X 105.778,Y 89.198,Z 74.580,A 180.000,B 0.000,C 180.000} C_DIS
LIN {X 105.722,Y 89.142,Z 74.577,A 180.000,B 0.000,C 180.000} C_DIS
LIN {X 105.666,Y 89.087,Z 74.575,A 180.000,B 0.000,C 180.000} C_DIS
LIN {X 105.554,Y 88.978,Z 74.570,A 180.000,B 0.000,C 180.000} C_DIS
LIN {X 105.441,Y 88.868,Z 74.565,A 180.000,B 0.000,C 180.000} C_DIS
LIN {X 105.328,Y 88.760,Z 74.560,A 180.000,B 0.000,C 180.000} C_DIS
LIN {X 105.210,Y 88.656,Z 74.556,A 180.000,B 0.000,C 180.000} C_DIS
LIN {X 105.091,Y 88.553,Z 74.551,A 180.000,B 0.000,C 180.000} C_DIS
LIN {X 104.972,Y 88.450,Z 74.547,A 180.000,B 0.000,C 180.000} C_DIS
LIN {X 104.852,Y 88.348,Z 74.543,A 180.000,B 0.000,C 180.000} C_DIS
LIN {X 104.731,Y 88.249,Z 74.539,A 180.000,B 0.000,C 180.000} C_DIS
LIN {X 104.606,Y 88.152,Z 74.535,A 180.000,B 0.000,C 180.000} C_DIS
LIN {X 104.481,Y 88.056,Z 74.532,A 180.000,B 0.000,C 180.000} C_DIS
LIN {X 104.356,Y 87.960,Z 74.528,A 180.000,B 0.000,C 180.000} C_DIS
LIN {X 104.228,Y 87.869,Z 74.525,A 180.000,B 0.000,C 180.000} C_DIS
LIN {X 104.098,Y 87.780,Z 74.522,A 180.000,B 0.000,C 180.000} C_DIS
LIN {X 103.968,Y 87.692,Z 74.519,A 180.000,B 0.000,C 180.000} C_DIS
LIN {X 103.838,Y 87.603,Z 74.516,A 180.000,B 0.000,C 180.000} C_DIS
LIN {X 103.706,Y 87.518,Z 74.514,A 180.000,B 0.000,C 180.000} C_DIS
LIN {X 103.436,Y 87.355,Z 74.509,A 180.000,B 0.000,C 180.000} C_DIS
LIN {X 103.164,Y 87.196,Z 74.506,A 180.000,B 0.000,C 180.000} C_DIS
LIN {X 102.885,Y 87.049,Z 74.503,A 180.000,B 0.000,C 180.000} C_DIS
LIN {X 102.605,Y 86.906,Z 74.501,A 180.000,B 0.000,C 180.000} C_DIS
LIN {X 102.318,Y 86.775,Z 74.500,A 180.000,B 0.000,C 180.000} C_DIS
LIN {X 102.191,Y 86.721,Z 74.500,A 180.000,B 0.000,C 180.000} C_DIS
; Cutting Move Starts
LIN {X 102.081,Y 86.672,Z 74.500,A 180.000,B 0.000,C 180.000} C_DIS
LIN {X 101.902,Y 86.597,Z 74.500,A 180.000,B 0.000,C 180.000} C_DIS
LIN {X 101.545,Y 86.461,Z 74.500,A 180.000,B 0.000,C 180.000} C_DIS
LIN {X 101.366,Y 86.396,Z 74.500,A 180.000,B 0.000,C 180.000} C_DIS
LIN {X 101.222,Y 86.349,Z 74.500,A 180.000,B 0.000,C 180.000} C_DIS
LIN {X 100.829,Y 86.224,Z 74.500,A 180.000,B 0.000,C 180.000} C_DIS
LIN {X 100.651,Y 86.172,Z 74.500,A 180.000,B 0.000,C 180.000} C_DIS
LIN {X 100.293,Y 86.080,Z 74.500,A 180.000,B 0.000,C 180.000} C_DIS
LIN {X 100.114,Y 86.036,Z 74.500,A 180.000,B 0.000,C 180.000} C_DIS
LIN {X 99.936,Y 86.000,Z 74.500,A 180.000,B 0.000,C 180.000} C_DIS
LIN {X 99.757,Y 85.964,Z 74.500,A 180.000,B 0.000,C 180.000} C_DIS
LIN {X 99.578,Y 85.929,Z 74.500,A 180.000,B 0.000,C 180.000} C_DIS
LIN {X 99.399,Y 85.896,Z 74.500,A 180.000,B 0.000,C 180.000} C_DIS
LIN {X 99.221,Y 85.871,Z 74.500,A 180.000,B 0.000,C 180.000} C_DIS
LIN {X 99.042,Y 85.845,Z 74.500,A 180.000,B 0.000,C 180.000} C_DIS
LIN {X 98.863,Y 85.820,Z 74.500,A 180.000,B 0.000,C 180.000} C_DIS
LIN {X 98.796,Y 85.813,Z 74.500,A 180.000,B 0.000,C 180.000} C_DIS
LIN {X 98.684,Y 85.803,Z 74.500,A 180.000,B 0.000,C 180.000} C_DIS
LIN {X 98.327,Y 85.773,Z 74.500,A 180.000,B 0.000,C 180.000} C_DIS
LIN {X 98.148,Y 85.760,Z 74.500,A 180.000,B 0.000,C 180.000} C_DIS
LIN {X 97.969,Y 85.753,Z 74.500,A 180.000,B 0.000,C 180.000} C_DIS
LIN {X 97.612,Y 85.743,Z 74.500,A 180.000,B 0.000,C 180.000} C_DIS
LIN {X 97.433,Y 85.742,Z 74.500,A 180.000,B 0.000,C 180.000} C_DIS
LIN {X 97.075,Y 85.752,Z 74.500,A 180.000,B 0.000,C 180.000} C_DIS
LIN {X 96.897,Y 85.758,Z 74.500,A 180.000,B 0.000,C 180.000} C_DIS
LIN {X 96.718,Y 85.769,Z 74.500,A 180.000,B 0.000,C 180.000} C_DIS
LIN {X 96.360,Y 85.799,Z 74.500,A 180.000,B 0.000,C 180.000} C_DIS
LIN {X 96.204,Y 85.813,Z 74.500,A 180.000,B 0.000,C 180.000} C_DIS
LIN {X 96.181,Y 85.815,Z 74.500,A 180.000,B 0.000,C 180.000} C_DIS
LIN {X 96.003,Y 85.839,Z 74.500,A 180.000,B 0.000,C 180.000} C_DIS
LIN {X 95.645,Y 85.890,Z 74.500,A 180.000,B 0.000,C 180.000} C_DIS
LIN {X 95.466,Y 85.920,Z 74.500,A 180.000,B 0.000,C 180.000} C_DIS
LIN {X 95.288,Y 85.955,Z 74.500,A 180.000,B 0.000,C 180.000} C_DIS
LIN {X 94.930,Y 86.026,Z 74.500,A 180.000,B 0.000,C 180.000} C_DIS
LIN {X 94.751,Y 86.068,Z 74.500,A 180.000,B 0.000,C 180.000} C_DIS
LIN {X 94.356,Y 86.170,Z 74.500,A 180.000,B 0.000,C 180.000} C_DIS
LIN {X 94.215,Y 86.210,Z 74.500,A 180.000,B 0.000,C 180.000} C_DIS
LIN {X 94.036,Y 86.267,Z 74.500,A 180.000,B 0.000,C 180.000} C_DIS
LIN {X 93.778,Y 86.349,Z 74.500,A 180.000,B 0.000,C 180.000} C_DIS
LIN {X 93.679,Y 86.381,Z 74.500,A 180.000,B 0.000,C 180.000} C_DIS
LIN {X 93.500,Y 86.444,Z 74.500,A 180.000,B 0.000,C 180.000} C_DIS
LIN {X 93.142,Y 86.580,Z 74.500,A 180.000,B 0.000,C 180.000} C_DIS
LIN {X 92.964,Y 86.652,Z 74.500,A 180.000,B 0.000,C 180.000} C_DIS
LIN {X 92.841,Y 86.707,Z 74.500,A 180.000,B 0.000,C 180.000} C_DIS
LIN {X 92.606,Y 86.812,Z 74.500,A 180.000,B 0.000,C 180.000} C_DIS
LIN {X 92.444,Y 86.885,Z 74.500,A 180.000,B 0.000,C 180.000} C_DIS
LIN {X 92.427,Y 86.893,Z 74.500,A 180.000,B 0.000,C 180.000} C_DIS
LIN {X 92.249,Y 86.981,Z 74.500,A 180.000,B 0.000,C 180.000} C_DIS
LIN {X 91.891,Y 87.166,Z 74.500,A 180.000,B 0.000,C 180.000} C_DIS
LIN {X 91.751,Y 87.243,Z 74.500,A 180.000,B 0.000,C 180.000} C_DIS
LIN {X 91.355,Y 87.477,Z 74.500,A 180.000,B 0.000,C 180.000} C_DIS
LIN {X 91.176,Y 87.588,Z 74.500,A 180.000,B 0.000,C 180.000} C_DIS
LIN {X 91.157,Y 87.601,Z 74.500,A 180.000,B 0.000,C 180.000} C_DIS
LIN {X 90.997,Y 87.707,Z 74.500,A 180.000,B 0.000,C 180.000} C_DIS
LIN {X 90.818,Y 87.827,Z 74.500,A 180.000,B 0.000,C 180.000} C_DIS
LIN {X 90.640,Y 87.950,Z 74.500,A 180.000,B 0.000,C 180.000} C_DIS
LIN {X 90.629,Y 87.958,Z 74.500,A 180.000,B 0.000,C 180.000} C_DIS
LIN {X 90.282,Y 88.219,Z 74.500,A 180.000,B 0.000,C 180.000} C_DIS
LIN {X 90.159,Y 88.316,Z 74.500,A 180.000,B 0.000,C 180.000} C_DIS
LIN {X 90.103,Y 88.362,Z 74.500,A 180.000,B 0.000,C 180.000} C_DIS
LIN {X 89.945,Y 88.494,Z 74.500,A 180.000,B 0.000,C 180.000} C_DIS
LIN {X 89.734,Y 88.673,Z 74.500,A 180.000,B 0.000,C 180.000} C_DIS
LIN {X 89.567,Y 88.822,Z 74.500,A 180.000,B 0.000,C 180.000} C_DIS
LIN {X 89.346,Y 89.031,Z 74.500,A 180.000,B 0.000,C 180.000} C_DIS
LIN {X 89.209,Y 89.161,Z 74.500,A 180.000,B 0.000,C 180.000} C_DIS
LIN {X 89.162,Y 89.209,Z 74.500,A 180.000,B 0.000,C 180.000} C_DIS
LIN {X 89.031,Y 89.349,Z 74.500,A 180.000,B 0.000,C 180.000} C_DIS
LIN {X 88.852,Y 89.538,Z 74.500,A 180.000,B 0.000,C 180.000} C_DIS
LIN {X 88.824,Y 89.567,Z 74.500,A 180.000,B 0.000,C 180.000} C_DIS
LIN {X 88.673,Y 89.732,Z 74.500,A 180.000,B 0.000,C 180.000} C_DIS
LIN {X 88.662,Y 89.746,Z 74.500,A 180.000,B 0.000,C 180.000} C_DIS
LIN {X 88.360,Y 90.103,Z 74.500,A 180.000,B 0.000,C 180.000} C_DIS
LIN {X 88.316,Y 90.157,Z 74.500,A 180.000,B 0.000,C 180.000} C_DIS
LIN {X 88.220,Y 90.282,Z 74.500,A 180.000,B 0.000,C 180.000} C_DIS
LIN {X 88.086,Y 90.461,Z 74.500,A 180.000,B 0.000,C 180.000} C_DIS
LIN {X 87.958,Y 90.631,Z 74.500,A 180.000,B 0.000,C 180.000} C_DIS
LIN {X 87.952,Y 90.640,Z 74.500,A 180.000,B 0.000,C 180.000} C_DIS
LIN {X 87.826,Y 90.818,Z 74.500,A 180.000,B 0.000,C 180.000} C_DIS
LIN {X 87.587,Y 91.176,Z 74.500,A 180.000,B 0.000,C 180.000} C_DIS
LIN {X 87.477,Y 91.355,Z 74.500,A 180.000,B 0.000,C 180.000} C_DIS
LIN {X 87.266,Y 91.712,Z 74.500,A 180.000,B 0.000,C 180.000} C_DIS
LIN {X 87.243,Y 91.752,Z 74.500,A 180.000,B 0.000,C 180.000} C_DIS
LIN {X 87.167,Y 91.891,Z 74.500,A 180.000,B 0.000,C 180.000} C_DIS
LIN {X 87.074,Y 92.070,Z 74.500,A 180.000,B 0.000,C 180.000} C_DIS
LIN {X 86.982,Y 92.249,Z 74.500,A 180.000,B 0.000,C 180.000} C_DIS
LIN {X 86.891,Y 92.427,Z 74.500,A 180.000,B 0.000,C 180.000} C_DIS
LIN {X 86.885,Y 92.440,Z 74.500,A 180.000,B 0.000,C 180.000} C_DIS
LIN {X 86.811,Y 92.606,Z 74.500,A 180.000,B 0.000,C 180.000} C_DIS
LIN {X 86.707,Y 92.839,Z 74.500,A 180.000,B 0.000,C 180.000} C_DIS
LIN {X 86.652,Y 92.964,Z 74.500,A 180.000,B 0.000,C 180.000} C_DIS
LIN {X 86.581,Y 93.142,Z 74.500,A 180.000,B 0.000,C 180.000} C_DIS
LIN {X 86.445,Y 93.500,Z 74.500,A 180.000,B 0.000,C 180.000} C_DIS
LIN {X 86.380,Y 93.679,Z 74.500,A 180.000,B 0.000,C 180.000} C_DIS
LIN {X 86.349,Y 93.774,Z 74.500,A 180.000,B 0.000,C 180.000} C_DIS
LIN {X 86.266,Y 94.036,Z 74.500,A 180.000,B 0.000,C 180.000} C_DIS
LIN {X 86.209,Y 94.215,Z 74.500,A 180.000,B 0.000,C 180.000} C_DIS
LIN {X 86.170,Y 94.362,Z 74.500,A 180.000,B 0.000,C 180.000} C_DIS
LIN {X 86.070,Y 94.751,Z 74.500,A 180.000,B 0.000,C 180.000} C_DIS
LIN {X 86.026,Y 94.930,Z 74.500,A 180.000,B 0.000,C 180.000} C_DIS
LIN {X 85.992,Y 95.099,Z 74.500,A 180.000,B 0.000,C 180.000} C_DIS
LIN {X 85.954,Y 95.288,Z 74.500,A 180.000,B 0.000,C 180.000} C_DIS
LIN {X 85.919,Y 95.466,Z 74.500,A 180.000,B 0.000,C 180.000} C_DIS
LIN {X 85.890,Y 95.645,Z 74.500,A 180.000,B 0.000,C 180.000} C_DIS
LIN {X 85.840,Y 96.003,Z 74.500,A 180.000,B 0.000,C 180.000} C_DIS
LIN {X 85.823,Y 96.133,Z 74.500,A 180.000,B 0.000,C 180.000} C_DIS
LIN {X 85.816,Y 96.181,Z 74.500,A 180.000,B 0.000,C 180.000} C_DIS
LIN {X 85.813,Y 96.210,Z 74.500,A 180.000,B 0.000,C 180.000} C_DIS
LIN {X 85.799,Y 96.360,Z 74.500,A 180.000,B 0.000,C 180.000} C_DIS
LIN {X 85.769,Y 96.718,Z 74.500,A 180.000,B 0.000,C 180.000} C_DIS
LIN {X 85.757,Y 96.897,Z 74.500,A 180.000,B 0.000,C 180.000} C_DIS
LIN {X 85.752,Y 97.075,Z 74.500,A 180.000,B 0.000,C 180.000} C_DIS
LIN {X 85.747,Y 97.254,Z 74.500,A 180.000,B 0.000,C 180.000} C_DIS
LIN {X 85.743,Y 97.433,Z 74.500,A 180.000,B 0.000,C 180.000} C_DIS
LIN {X 85.743,Y 97.612,Z 74.500,A 180.000,B 0.000,C 180.000} C_DIS
LIN {X 85.748,Y 97.790,Z 74.500,A 180.000,B 0.000,C 180.000} C_DIS
LIN {X 85.753,Y 97.969,Z 74.500,A 180.000,B 0.000,C 180.000} C_DIS
LIN {X 85.759,Y 98.148,Z 74.500,A 180.000,B 0.000,C 180.000} C_DIS
LIN {X 85.772,Y 98.327,Z 74.500,A 180.000,B 0.000,C 180.000} C_DIS
LIN {X 85.803,Y 98.684,Z 74.500,A 180.000,B 0.000,C 180.000} C_DIS
LIN {X 85.813,Y 98.790,Z 74.500,A 180.000,B 0.000,C 180.000} C_DIS
LIN {X 85.822,Y 98.863,Z 74.500,A 180.000,B 0.000,C 180.000} C_DIS
LIN {X 85.846,Y 99.042,Z 74.500,A 180.000,B 0.000,C 180.000} C_DIS
LIN {X 85.897,Y 99.399,Z 74.500,A 180.000,B 0.000,C 180.000} C_DIS
LIN {X 85.927,Y 99.578,Z 74.500,A 180.000,B 0.000,C 180.000} C_DIS
LIN {X 85.998,Y 99.936,Z 74.500,A 180.000,B 0.000,C 180.000} C_DIS
LIN {X 86.036,Y 100.114,Z 74.500,A 180.000,B 0.000,C 180.000} C_DIS
LIN {X 86.081,Y 100.293,Z 74.500,A 180.000,B 0.000,C 180.000} C_DIS
LIN {X 86.174,Y 100.651,Z 74.500,A 180.000,B 0.000,C 180.000} C_DIS
LIN {X 86.223,Y 100.829,Z 74.500,A 180.000,B 0.000,C 180.000} C_DIS
LIN {X 86.280,Y 101.008,Z 74.500,A 180.000,B 0.000,C 180.000} C_DIS
LIN {X 86.349,Y 101.226,Z 74.500,A 180.000,B 0.000,C 180.000} C_DIS
LIN {X 86.395,Y 101.366,Z 74.500,A 180.000,B 0.000,C 180.000} C_DIS
LIN {X 86.462,Y 101.545,Z 74.500,A 180.000,B 0.000,C 180.000} C_DIS
LIN {X 86.530,Y 101.723,Z 74.500,A 180.000,B 0.000,C 180.000} C_DIS
LIN {X 86.598,Y 101.902,Z 74.500,A 180.000,B 0.000,C 180.000} C_DIS
LIN {X 86.671,Y 102.081,Z 74.500,A 180.000,B 0.000,C 180.000} C_DIS
LIN {X 86.707,Y 102.161,Z 74.500,A 180.000,B 0.000,C 180.000} C_DIS
LIN {X 86.831,Y 102.438,Z 74.500,A 180.000,B 0.000,C 180.000} C_DIS
LIN {X 86.885,Y 102.560,Z 74.500,A 180.000,B 0.000,C 180.000} C_DIS
LIN {X 86.913,Y 102.617,Z 74.500,A 180.000,B 0.000,C 180.000} C_DIS
LIN {X 87.005,Y 102.796,Z 74.500,A 180.000,B 0.000,C 180.000} C_DIS
LIN {X 87.097,Y 102.975,Z 74.500,A 180.000,B 0.000,C 180.000} C_DIS
LIN {X 87.191,Y 103.153,Z 74.500,A 180.000,B 0.000,C 180.000} C_DIS
LIN {X 87.243,Y 103.248,Z 74.500,A 180.000,B 0.000,C 180.000} C_DIS
LIN {X 87.292,Y 103.332,Z 74.500,A 180.000,B 0.000,C 180.000} C_DIS
LIN {X 87.503,Y 103.690,Z 74.500,A 180.000,B 0.000,C 180.000} C_DIS
LIN {X 87.601,Y 103.844,Z 74.500,A 180.000,B 0.000,C 180.000} C_DIS
LIN {X 87.779,Y 104.111,Z 74.500,A 180.000,B 0.000,C 180.000} C_DIS
LIN {X 87.856,Y 104.226,Z 74.500,A 180.000,B 0.000,C 180.000} C_DIS
LIN {X 87.958,Y 104.369,Z 74.500,A 180.000,B 0.000,C 180.000} C_DIS
LIN {X 87.985,Y 104.405,Z 74.500,A 180.000,B 0.000,C 180.000} C_DIS
LIN {X 88.254,Y 104.762,Z 74.500,A 180.000,B 0.000,C 180.000} C_DIS
LIN {X 88.316,Y 104.843,Z 74.500,A 180.000,B 0.000,C 180.000} C_DIS
LIN {X 88.397,Y 104.941,Z 74.500,A 180.000,B 0.000,C 180.000} C_DIS
LIN {X 88.548,Y 105.120,Z 74.500,A 180.000,B 0.000,C 180.000} C_DIS
LIN {X 88.673,Y 105.268,Z 74.500,A 180.000,B 0.000,C 180.000} C_DIS
LIN {X 88.700,Y 105.299,Z 74.500,A 180.000,B 0.000,C 180.000} C_DIS
LIN {X 88.852,Y 105.462,Z 74.500,A 180.000,B 0.000,C 180.000} C_DIS
LIN {X 89.035,Y 105.656,Z 74.500,A 180.000,B 0.000,C 180.000} C_DIS
LIN {X 89.206,Y 105.835,Z 74.500,A 180.000,B 0.000,C 180.000} C_DIS
LIN {X 89.209,Y 105.839,Z 74.500,A 180.000,B 0.000,C 180.000} C_DIS
LIN {X 89.388,Y 106.009,Z 74.500,A 180.000,B 0.000,C 180.000} C_DIS
LIN {X 89.583,Y 106.193,Z 74.500,A 180.000,B 0.000,C 180.000} C_DIS
LIN {X 89.746,Y 106.337,Z 74.500,A 180.000,B 0.000,C 180.000} C_DIS
LIN {X 89.998,Y 106.550,Z 74.500,A 180.000,B 0.000,C 180.000} C_DIS
LIN {X 90.103,Y 106.638,Z 74.500,A 180.000,B 0.000,C 180.000} C_DIS
LIN {X 90.214,Y 106.729,Z 74.500,A 180.000,B 0.000,C 180.000} C_DIS
LIN {X 90.282,Y 106.781,Z 74.500,A 180.000,B 0.000,C 180.000} C_DIS
LIN {X 90.461,Y 106.915,Z 74.500,A 180.000,B 0.000,C 180.000} C_DIS
LIN {X 90.640,Y 107.050,Z 74.500,A 180.000,B 0.000,C 180.000} C_DIS
LIN {X 90.690,Y 107.086,Z 74.500,A 180.000,B 0.000,C 180.000} C_DIS
LIN {X 90.818,Y 107.173,Z 74.500,A 180.000,B 0.000,C 180.000} C_DIS
LIN {X 90.997,Y 107.293,Z 74.500,A 180.000,B 0.000,C 180.000} C_DIS
LIN {X 91.176,Y 107.412,Z 74.500,A 180.000,B 0.000,C 180.000} C_DIS
LIN {X 91.227,Y 107.444,Z 74.500,A 180.000,B 0.000,C 180.000} C_DIS
LIN {X 91.355,Y 107.523,Z 74.500,A 180.000,B 0.000,C 180.000} C_DIS
LIN {X 91.712,Y 107.734,Z 74.500,A 180.000,B 0.000,C 180.000} C_DIS
LIN {X 91.829,Y 107.802,Z 74.500,A 180.000,B 0.000,C 180.000} C_DIS
LIN {X 91.891,Y 107.834,Z 74.500,A 180.000,B 0.000,C 180.000} C_DIS
LIN {X 92.249,Y 108.019,Z 74.500,A 180.000,B 0.000,C 180.000} C_DIS
LIN {X 92.427,Y 108.107,Z 74.500,A 180.000,B 0.000,C 180.000} C_DIS
LIN {X 92.541,Y 108.159,Z 74.500,A 180.000,B 0.000,C 180.000} C_DIS
LIN {X 92.940,Y 108.338,Z 74.500,A 180.000,B 0.000,C 180.000} C_DIS
LIN {X 92.964,Y 108.348,Z 74.500,A 180.000,B 0.000,C 180.000} C_DIS
LIN {X 93.142,Y 108.420,Z 74.500,A 180.000,B 0.000,C 180.000} C_DIS
LIN {X 93.500,Y 108.556,Z 74.500,A 180.000,B 0.000,C 180.000} C_DIS
LIN {X 93.679,Y 108.619,Z 74.500,A 180.000,B 0.000,C 180.000} C_DIS
LIN {X 93.857,Y 108.676,Z 74.500,A 180.000,B 0.000,C 180.000} C_DIS
LIN {X 94.036,Y 108.733,Z 74.500,A 180.000,B 0.000,C 180.000} C_DIS
LIN {X 94.215,Y 108.790,Z 74.500,A 180.000,B 0.000,C 180.000} C_DIS
LIN {X 94.394,Y 108.839,Z 74.500,A 180.000,B 0.000,C 180.000} C_DIS
LIN {X 94.751,Y 108.932,Z 74.500,A 180.000,B 0.000,C 180.000} C_DIS
LIN {X 94.930,Y 108.974,Z 74.500,A 180.000,B 0.000,C 180.000} C_DIS
LIN {X 95.328,Y 109.053,Z 74.500,A 180.000,B 0.000,C 180.000} C_DIS
LIN {X 95.466,Y 109.080,Z 74.500,A 180.000,B 0.000,C 180.000} C_DIS
LIN {X 95.645,Y 109.110,Z 74.500,A 180.000,B 0.000,C 180.000} C_DIS
LIN {X 96.003,Y 109.161,Z 74.500,A 180.000,B 0.000,C 180.000} C_DIS
LIN {X 96.181,Y 109.185,Z 74.500,A 180.000,B 0.000,C 180.000} C_DIS
LIN {X 96.360,Y 109.201,Z 74.500,A 180.000,B 0.000,C 180.000} C_DIS
LIN {X 96.718,Y 109.231,Z 74.500,A 180.000,B 0.000,C 180.000} C_DIS
LIN {X 96.728,Y 109.232,Z 74.500,A 180.000,B 0.000,C 180.000} C_DIS
LIN {X 96.897,Y 109.242,Z 74.500,A 180.000,B 0.000,C 180.000} C_DIS
LIN {X 97.075,Y 109.248,Z 74.500,A 180.000,B 0.000,C 180.000} C_DIS
LIN {X 97.433,Y 109.258,Z 74.500,A 180.000,B 0.000,C 180.000} C_DIS
LIN {X 97.612,Y 109.257,Z 74.500,A 180.000,B 0.000,C 180.000} C_DIS
LIN {X 97.969,Y 109.247,Z 74.500,A 180.000,B 0.000,C 180.000} C_DIS
LIN {X 98.148,Y 109.240,Z 74.500,A 180.000,B 0.000,C 180.000} C_DIS
LIN {X 98.272,Y 109.232,Z 74.500,A 180.000,B 0.000,C 180.000} C_DIS
